// TwinCAT 3 PLC project LULSolarData
// ProgramVersion: 3.1.4020.10
// libraries:
//   Tc2_BA, * (Beckhoff Automation GmbH)
//   Tc2_EtherCAT, * (Beckhoff Automation GmbH)
//   Tc2_IoFunctions, * (Beckhoff Automation GmbH)
//   Tc2_ModbusRTU, * (Beckhoff Automation GmbH)
//   Tc2_ModbusSrv, * (Beckhoff Automation GmbH)
//   Tc2_SerialCom, * (Beckhoff Automation GmbH)
//   Tc2_Standard, * (Beckhoff Automation GmbH)
//   Tc2_SUPS, * (Beckhoff Automation GmbH)
//   Tc2_System, * (Beckhoff Automation GmbH)
//   Tc2_Utilities, * (Beckhoff Automation GmbH)
//   Tc3_IotBase, * (Beckhoff Automation GmbH)
//   Tc3_Module, * (Beckhoff Automation GmbH)
// project tree:
//   DUTs/Cluster Control/Huvudstrukt/ ST_ClusterCtrl.TcDUT
//   DUTs/Cluster Control/ ST_ActivePower.TcDUT, ST_ApparentPower.TcDUT, ST_DcCurrent.TcDUT, ST_LineCurrent.TcDUT, ST_LineVoltage.TcDUT, ST_PV_data.TcDUT, ST_ReactivePower.TcDUT, ST_Si420TC.TcDUT, ST_StatusCtrl.TcDUT, ST_Yield.TcDUT
//   DUTs/Hukseflux SR05/ ST_SR05_IrrMeter.TcDUT
//   DUTs/IoT/ U_Payload.TcDUT
//   DUTs/Schneider IEM/Huvudstrukt/ ST_IEM3255.TcDUT
//   DUTs/Schneider IEM/ ST_AlarmValue.TcDUT, ST_OverloadAL.TcDUT, ST_Current.TcDUT, ST_Frequency.TcDUT, ST_PartialEnergy.TcDUT, ST_PhaseEnergy.TcDUT, ST_Power.TcDUT, ST_Power2.TcDUT, ST_PowerFactor.TcDUT, ST_TotalEnergy.TcDUT, ST_Voltage.TcDUT, ST_Voltage2.TcDUT
//   DUTs/WXT530/Huvudstrukt/ ST_WXT530.TcDUT
//   DUTs/WXT530/ ST_WindData.TcDUT
//   GVLs/ GVL_ClusterCtrl.TcGVL, GVL_Fastighet.TcGVL, GVL_IO.TcGVL, GVL_IoT.TcGVL, GVL_Larm.TcGVL, GVL_MX41.TcGVL, GVL_SR05.TcGVL, GVL_WXT530.TcGVL
//   / Modbus.TcTTO, PlcTask.TcTTO
//   POUs/ClusterCtrl/ F15_ClusterCtrl.TcPOU, F15_ClusterCtrl_Larm.TcPOU
//   POUs/IO/ F15_AS3_AI.TcPOU
//   POUs/Loggning/ Cluster_Logg.TcPOU, Cluster_Logg_2.TcPOU, Cluster_Logg_3.TcPOU, Cluster_Sensor_Logg.TcPOU, FB_IoT_Publisher.TcPOU, iEM3255_Logg.TcPOU, MAIN_loggning.TcPOU, Temp_Logg.TcPOU, SR05_Logg.TcPOU, WXT530_Logg.TcPOU
//   POUs/ MAIN.TcPOU
//   POUs/MQ41/ F15_AS3_MQ41.TcPOU
//   POUs/Novram Hantering/ NovramHandling.TcPOU
//   POUs/Novram Hantering/ST_Novram/ ST_NovramData.TcDUT
//   POUs/Systemprogram/ PersistentData.TcPOU, PLC_Batteri_Larm.TcPOU, PLC_TID.TcPOU, WatchDog_PLC.TcPOU
//   POUs/WXT530/ F15_AS3_WXT530.TcPOU, RS485.TcPOU
//   POUs/_FBs/ AI_filter.TcPOU, ClusterControl_3Unit.TcPOU, FB_CountYears.TcPOU, FB_FL.TcPOU, FB_Pulsfilter.TcPOU, FB_SaveToCSV_ClusterCtrl.TcPOU, FB_SaveToCSV_SR05.TcPOU, FB_SaveToCSV_Schneider.TcPOU, FB_SaveToCSV_Cluster_Sensors.TcPOU, FB_SaveToCSV_Temp.TcPOU, FB_SaveToCSV_WXT530.TcPOU, FB_SCHNEIDER_iEM3150.TcPOU, FB_HUKSEFLUX_SR05.TcPOU, FB_WXT350.TcPOU, F_WordSwap.TcPOU
// real-time tasks:
//   TASK PlcTask: cycle T#5ms, priority 3, ADS port 350
//   TASK Modbus_seriell: cycle T#1ms, priority 1, ADS port 352
// I/O:
//   DEVICE Device 1 (EtherCAT), AmsNetId 172.17.204.1.2.1
//     Term 5 (EK1200) [EK1200-5000 EtherCAT Power supply (2A E-Bus)]
//       Term 6 (EL6021) [EL6021 Interface (RS422/485)]
//       Term 7 (EL6021) [EL6021 Interface (RS422/485)]
//       Box 8 (BK1250)
//   DEVICE Device 5 (USB) (disabled)
//   DEVICE Device 6 (NOV-DP-RAM)
// variable links:
//   LULSolarData/LULSolarData Instance <-> Device 1 (EtherCAT)/Term 5 (EK1200)/Box 8 (BK1250)
//     PlcTask Inputs/GVL_IO._AI1 <-> Term 2 (KL3208-0010-4)/Channel 1/Data In
//     PlcTask Inputs/GVL_IO._AI2 <-> Term 2 (KL3208-0010-4)/Channel 2/Data In
//     PlcTask Inputs/GVL_IO._AI3 <-> Term 2 (KL3208-0010-4)/Channel 3/Data In
//     PlcTask Inputs/GVL_IO._AI4 <-> Term 2 (KL3208-0010-4)/Channel 4/Data In
//     PlcTask Inputs/GVL_IO._AI5 <-> Term 3 (KL3208-0010-4)/Channel 1/Data In
//     PlcTask Inputs/GVL_IO._AI6 <-> Term 3 (KL3208-0010-4)/Channel 2/Data In
//     PlcTask Inputs/GVL_IO._AI7 <-> Term 3 (KL3208-0010-4)/Channel 3/Data In
//     PlcTask Inputs/GVL_IO._AI8 <-> Term 3 (KL3208-0010-4)/Channel 4/Data In
//   LULSolarData/LULSolarData Instance <-> Device 1 (EtherCAT)/Term 5 (EK1200)/Term 6 (EL6021)
//     Modbus Inputs/RS485.ComIn_Com1/D <-> COM TxPDO-Map Inputs/Data In 0
//     Modbus Inputs/RS485.ComIn_Com1/D @bit {8..168 step 8} <-> COM TxPDO-Map Inputs/Data In {1..21}  (21 links)
//     Modbus Inputs/RS485.ComIn_Com1/Status <-> COM TxPDO-Map Inputs/Status
//     Modbus Outputs/RS485.ComOut_Com1/Ctrl <-> COM RxPDO-Map Outputs/Ctrl
//     Modbus Outputs/RS485.ComOut_Com1/D <-> COM RxPDO-Map Outputs/Data Out 0
//     Modbus Outputs/RS485.ComOut_Com1/D @bit {8..168 step 8} <-> COM RxPDO-Map Outputs/Data Out {1..21}  (21 links)
//   LULSolarData/LULSolarData Instance <-> Device 1 (EtherCAT)/Term 5 (EK1200)/Term 7 (EL6021)
//     Modbus Inputs/F15_AS3_MQ41.Energimatare.fbRtuMaster.InData/D <-> COM TxPDO-Map Inputs/Data In 0
//     Modbus Inputs/F15_AS3_MQ41.Energimatare.fbRtuMaster.InData/D @bit {8..168 step 8} <-> COM TxPDO-Map Inputs/Data In {1..21}  (21 links)
//     Modbus Inputs/F15_AS3_MQ41.Energimatare.fbRtuMaster.InData/Status <-> COM TxPDO-Map Inputs/Status
//     Modbus Outputs/F15_AS3_MQ41.Energimatare.fbRtuMaster.OutData/Ctrl <-> COM RxPDO-Map Outputs/Ctrl
//     Modbus Outputs/F15_AS3_MQ41.Energimatare.fbRtuMaster.OutData/D <-> COM RxPDO-Map Outputs/Data Out 0
//     Modbus Outputs/F15_AS3_MQ41.Energimatare.fbRtuMaster.OutData/D @bit {8..168 step 8} <-> COM RxPDO-Map Outputs/Data Out {1..21}  (21 links)

CONFIGURATION LULSolarData
    RESOURCE PLC ON TwinCAT3
        TASK Modbus(INTERVAL := T#1ms, PRIORITY := 1);
        TASK PlcTask(INTERVAL := T#5ms, PRIORITY := 3);
        PROGRAM F15_AS3_MQ41 WITH Modbus : F15_AS3_MQ41;
        PROGRAM F15_AS3_WXT530 WITH Modbus : F15_AS3_WXT530;
        PROGRAM RS485 WITH Modbus : RS485;
        PROGRAM MAIN WITH PlcTask : MAIN;
    END_RESOURCE
END_CONFIGURATION

// ---- DUTs/Cluster Control/Huvudstrukt/ST_ClusterCtrl.TcDUT
TYPE ST_ClusterCtrl :
STRUCT
	stActivePower			:ST_ActivePower;
	stLineVoltage			:ST_LineVoltage;
	stLineCurrent			:ST_LineCurrent;
	stYield					:ST_Yield;
	stPVDATA				:ST_PV_data;
	stStatus				:ST_StatusCtrl;
	stReactivePower			:ST_ReactivePower;
	stApparentPower			:ST_ApparentPower;
	stSi420					:ST_Si420TC;
	nTotEnergyConsInternally:DWORD;
	nInverterInteriorTemp 	:DWORD;
	nEnergySavingMode		:DWORD;
END_STRUCT
END_TYPE

// ---- DUTs/Cluster Control/ST_ActivePower.TcDUT
TYPE ST_ActivePower :
STRUCT
	
	ActivePower_Total		:DINT;
	ActivePower_L1			:DINT;
	ActivePower_L2			:DINT;
	ActivePower_L3			:DINT;
	
END_STRUCT
END_TYPE

// ---- DUTs/Cluster Control/ST_ApparentPower.TcDUT
TYPE ST_ApparentPower :
STRUCT
	ApparentPower_Total			:DINT;
	ApparentPower_L1			:DINT;
	ApparentPower_L2			:DINT;
	ApparentPower_L3			:DINT;
END_STRUCT
END_TYPE

// ---- DUTs/Cluster Control/ST_DcCurrent.TcDUT
TYPE ST_DcCurrent :
STRUCT
	
END_STRUCT
END_TYPE

// ---- DUTs/Cluster Control/ST_LineCurrent.TcDUT
TYPE ST_LineCurrent :
STRUCT
	
	LineCurrent_Total		:DWORD;
	LineCurrent_L1			:DWORD;
	LineCurrent_L2			:DWORD;
	LineCurrent_L3			:DWORD;
	PowerFrequency			:DWORD;
	
END_STRUCT
END_TYPE

// ---- DUTs/Cluster Control/ST_LineVoltage.TcDUT
TYPE ST_LineVoltage :
STRUCT
	
	LineVoltage_L1_N 	:DWORD;
	LineVoltage_L2_N 	:DWORD;
	LineVoltage_L3_N 	:DWORD;
	LineVoltage_L1_L2 	:DWORD;
	LineVoltage_L2_L3 	:DWORD;
	LineVoltage_L3_L1 	:DWORD;
	
END_STRUCT
END_TYPE

// ---- DUTs/Cluster Control/ST_PV_data.TcDUT
TYPE ST_PV_data :
STRUCT
	Line_current_L1		:DINT;
	Line_current_L2		:DINT;
	Line_current_L3		:DINT;
	PV_Power			:DWORD;
END_STRUCT
END_TYPE

// ---- DUTs/Cluster Control/ST_ReactivePower.TcDUT
TYPE ST_ReactivePower :
STRUCT
	ReactivePower_Total		:DINT;
	ReactivePower_L1		:DINT;
	ReactivePower_L2		:DINT;
	ReactivePower_L3		:DINT;
END_STRUCT
END_TYPE

// ---- DUTs/Cluster Control/ST_Si420TC.TcDUT
TYPE ST_Si420TC :
STRUCT
	Irradiation	:DINT;
END_STRUCT
END_TYPE

// ---- DUTs/Cluster Control/ST_StatusCtrl.TcDUT
TYPE ST_StatusCtrl :
STRUCT
	Device_Status		:DWORD;
END_STRUCT
END_TYPE

// ---- DUTs/Cluster Control/ST_Yield.TcDUT
TYPE ST_Yield :
STRUCT
	Total_AC_energy_all_conductors_Wh		:DWORD;
	Total_AC_energy_all_conductors_kWh		:DWORD;
	Total_AC_energy_all_conductors_MWh		:DWORD;
	Energy_current_day_all_conductors_Wh	:DWORD;
	Energy_current_day_all_conductors_kWh	:DWORD;
	Energy_current_day_all_conductors_MWh	:DWORD;
	Operating_time							:DWORD;
	Feed_in_time							:DWORD;	
END_STRUCT
END_TYPE

// ---- DUTs/Hukseflux SR05/ST_SR05_IrrMeter.TcDUT
TYPE ST_SR05_IrrMeter :
STRUCT
	Solar_Irradiance_raw:  		REAL;
	Solar_Irradiance:   		REAL;
	Sensor_Body_Temp:			REAL;
	Sensor_Elec_Resistance:		REAL;
	Sensor_voltage_output:		REAL;
	
END_STRUCT
END_TYPE

// ---- DUTs/IoT/U_Payload.TcDUT
TYPE U_Payload :
UNION
	sPayload : STRING(3999);
	aPayload : ARRAY[0..3999] OF BYTE;
END_UNION
END_TYPE

// ---- DUTs/Schneider IEM/Huvudstrukt/ST_IEM3255.TcDUT
TYPE ST_IEM3255 :
STRUCT
	stCurrent:			ST_Current;
	stVolt:				ST_Voltage;
	stVolt2:			ST_Voltage2;
	stPower:			ST_Power;
	stPower2:			ST_Power2;
	stPowerFactor:		ST_PowerFactor;
	stFrequency:		ST_Frequency;
	stTotalEnergy:		ST_TotalEnergy;
	stPartialEnergy:	ST_PartialEnergy;
	stPhaseEnergy:		ST_PhaseEnergy;
	stOverloadAL:		ST_OverloadAL;
	stAlarmValue:		ST_AlarmValue;
END_STRUCT
END_TYPE

// ---- DUTs/Schneider IEM/ST_AlarmValue.TcDUT
TYPE ST_AlarmValue :
STRUCT
	Last_Alarm_Value:	REAL;
END_STRUCT
END_TYPE

// ---- DUTs/Schneider IEM/ST_OverloadAL.TcDUT
TYPE ST_OverloadAL :
STRUCT
	Status:	BIT;
END_STRUCT
END_TYPE

// ---- DUTs/Schneider IEM/ST_Current.TcDUT
TYPE ST_Current :
STRUCT
	Phase_1_current:	REAL;
	Phase_2_current:	REAL;
	Phase_3_current:	REAL;
END_STRUCT
END_TYPE

// ---- DUTs/Schneider IEM/ST_Frequency.TcDUT
TYPE ST_Frequency :
STRUCT
	Frequency:	REAL;
END_STRUCT
END_TYPE

// ---- DUTs/Schneider IEM/ST_PartialEnergy.TcDUT
TYPE ST_PartialEnergy :
STRUCT
	Partial_Active_Energy_Import:	REAL;
	Partial_Reactive_Energy_Import:	REAL;
END_STRUCT
END_TYPE

// ---- DUTs/Schneider IEM/ST_PhaseEnergy.TcDUT
TYPE ST_PhaseEnergy :
STRUCT
	Active_Energy_Import_Phase_1:	REAL;
	Active_Energy_Import_Phase_2:	REAL;
	Active_Energy_Import_Phase_3:	REAL;
END_STRUCT
END_TYPE

// ---- DUTs/Schneider IEM/ST_Power.TcDUT
TYPE ST_Power :
STRUCT
	Active_Power_Phase_1:	REAL;
	Active_Power_Phase_2:	REAL;
	Active_Power_Phase_3:	REAL;
	Total_Active_Power:		REAL;
END_STRUCT
END_TYPE

// ---- DUTs/Schneider IEM/ST_Power2.TcDUT
TYPE ST_Power2 :
STRUCT
	Total_Reactive_Power:	REAL;
	Reserved2:				REAL;
	Reserved3:				REAL;
	Reserved4:				REAL;
	Total_Apparent_Power:	REAL;

END_STRUCT
END_TYPE

// ---- DUTs/Schneider IEM/ST_PowerFactor.TcDUT
TYPE ST_PowerFactor :
STRUCT
	Total_Power_Factor:	REAL;
END_STRUCT
END_TYPE

// ---- DUTs/Schneider IEM/ST_TotalEnergy.TcDUT
TYPE ST_TotalEnergy :
STRUCT
	Total_Active_Energy_Import:		REAL;
	Total_Active_Energy_Export:		REAL;
	Total_Reactive_Energy_Import:	REAL;
	Total_Reactive_Energy_Export:	REAL;
END_STRUCT
END_TYPE

// ---- DUTs/Schneider IEM/ST_Voltage.TcDUT
TYPE ST_Voltage :
STRUCT
	Voltage_L1_L2:	REAL;
	Voltage_L2_L3:	REAL;
	Voltage_L3_L1:	REAL;	
END_STRUCT
END_TYPE

// ---- DUTs/Schneider IEM/ST_Voltage2.TcDUT
TYPE ST_Voltage2 :
STRUCT
	Voltage_L1_N:	REAL;
	Voltage_L2_N:	REAL;
	Voltage_L3_N:	REAL;
END_STRUCT
END_TYPE

// ---- DUTs/WXT530/Huvudstrukt/ST_WXT530.TcDUT
TYPE ST_WXT530 :
STRUCT
	stWindData			:ST_WindData;
END_STRUCT
END_TYPE

// ---- DUTs/WXT530/ST_WindData.TcDUT
TYPE ST_WindData :
STRUCT

Dn	:REAL;  (*Wind direction minimum (D = degrees)*)
Dm	:REAL;  (*Wind direction average (D = degrees)*)
Dx	:REAL;  (*Wind direction maximum (D = degrees*)
Sn	:REAL;  (*Wind speed minimum (M = m/S)*)
Sm	:REAL;  (*Wind speed average (M = m/S)*)
Sx	:REAL;  (*Wind speed maximum (M = m/S)*)	

END_STRUCT
END_TYPE

// ---- POUs/Novram Hantering/ST_Novram/ST_NovramData.TcDUT
TYPE ST_NovramData :
STRUCT
END_STRUCT
END_TYPE

// ---- GVLs/GVL_ClusterCtrl.TcGVL
{attribute 'qualified_only'}
VAR_GLOBAL	
		
_CCtrl_V1_IT				AT%MX2000.0			:BOOL;  	(* Driftindikering *)
_CCtrl_V1_P					AT%MB2004			:REAL;  	(* Total momentan effekt *)
_CCtrl_V1_P1				AT%MB2008			:REAL;  	(* Effekt L1 *)
_CCtrl_V1_P2				AT%MB2012			:REAL;  	(* Effekt L2 *)
_CCtrl_V1_P3				AT%MB2016			:REAL;  	(* Effekt L3 *)
_CCtrl_V1_U1_L1_N			AT%MB2020			:REAL;  	(* Spänning L1-N *)
_CCtrl_V1_U2_L2_N			AT%MB2024			:REAL;  	(* Spänning L2-N *)
_CCtrl_V1_U3_L3_N			AT%MB2028			:REAL;  	(* Spänning L3-N *)
_CCtrl_V1_U1_L1_L2			AT%MB2032			:REAL;  	(* Spänning L1-L2*)
_CCtrl_V1_U2_L2_L3			AT%MB2036			:REAL;  	(* Spänning L2-L3 *)
_CCtrl_V1_U3_L3_L1			AT%MB2040			:REAL;  	(* Spänning L3-L1 *)
_CCtrl_V1_Itot									:REAL; 		(* Total Ström L1,L2,L3*)
_CCtrl_V1_I1				AT%MB2044			:REAL;  	(* Ström L1 *)
_CCtrl_V1_I2				AT%MB2048			:REAL;  	(* Ström L2 *)
_CCtrl_V1_I3				AT%MB2052			:REAL;  	(* Ström L3 *)
_CCtrl_V1_Yield_Wh			AT%MB2056			:REAL;  	(* Total avkastning Wh *)
_CCtrl_V1_Yield_kWh			AT%MB2060			:REAL;  	(* Total avkastning kWh *)
_CCtrl_V1_Yield_MWh			AT%MB2064			:REAL;  	(* Total avkastning MWh *)
_CCtrl_V1_YieldDay_Wh		AT%MB2068			:REAL;  	(* Total avkastning aktuell dag Wh *)
_CCtrl_V1_YieldDay_kWh		AT%MB2072			:REAL;  	(* Total avkastning aktuell dag kWh *)
_CCtrl_V1_PV				AT%MB2076			:REAL;  	(* PV effekt*)
_CCtrl_V1_HZ				AT%MB2080			:REAL;  	(* Frekvens *)	
_CCtrl_V1_TECInt								:REAL;		(* Total Energy Consumed Internally i växelriktaren *)	
_CCtrl_V1_APtot									:REAL;		(* Total Apparent Power L1,L2,L3*)
_CCtrl_V1_AP1									:REAL;  	(* Apparent Power L1 *)
_CCtrl_V1_AP2									:REAL;  	(* Apparent Power L2 *)
_CCtrl_V1_AP3									:REAL;  	(* Apparent Power L3 *)
_CCtrl_V1_RPtot									:REAL;		(* Total Reactive Power L1,L2,L3*)
_CCtrl_V1_RP1									:REAL;  	(* Reactive Power L1 *)
_CCtrl_V1_RP2									:REAL;  	(* Reactive Power L2 *)
_CCtrl_V1_RP3									:REAL;  	(* Reactive Power L3 *)
_CCtrl_V1_EnSaveMode							:REAL;		(* Energy Saving Mode Switched On (1129=Yes, 1130=No) *)

							
_CCtrl_V2_IT				AT%MX2400.0			:BOOL;  	(* Driftindikering *)
_CCtrl_V2_P					AT%MB2404			:REAL;  	(* Total momentan effekt *)
_CCtrl_V2_P1				AT%MB2408			:REAL;  	(* Effekt L1 *)
_CCtrl_V2_P2				AT%MB2412			:REAL;  	(* Effekt L2 *)
_CCtrl_V2_P3				AT%MB2416			:REAL;  	(* Effekt L3 *)
_CCtrl_V2_U1_L1_N			AT%MB2420			:REAL;  	(* Spänning L1-N *)
_CCtrl_V2_U2_L2_N			AT%MB2424			:REAL;  	(* Spänning L2-N *)
_CCtrl_V2_U3_L3_N			AT%MB2428			:REAL;  	(* Spänning L3-N *)
_CCtrl_V2_U1_L1_L2			AT%MB2432			:REAL;  	(* Spänning L1-L2*)
_CCtrl_V2_U2_L2_L3			AT%MB2436			:REAL;  	(* Spänning L2-L3 *)
_CCtrl_V2_U3_L3_L1			AT%MB2440			:REAL;  	(* Spänning L3-L1 *)
_CCtrl_V2_Itot									:REAL; 		(* Total Ström L1,L2,L3*)
_CCtrl_V2_I1				AT%MB2444			:REAL;  	(* Ström L1 *)
_CCtrl_V2_I2				AT%MB2448			:REAL;  	(* Ström L2 *)
_CCtrl_V2_I3				AT%MB2452			:REAL;  	(* Ström L3 *)
_CCtrl_V2_Yield_Wh			AT%MB2456			:REAL;  	(* Total avkastning Wh *)
_CCtrl_V2_Yield_kWh			AT%MB2460			:REAL;  	(* Total avkastning kWh *)
_CCtrl_V2_Yield_MWh			AT%MB2464			:REAL;  	(* Total avkastning MWh *)
_CCtrl_V2_YieldDay_Wh		AT%MB2468			:REAL;  	(* Total avkastning aktuell dag Wh *)
_CCtrl_V2_YieldDay_kWh		AT%MB2472			:REAL;  	(* Total avkastning aktuell dag kWh *)
_CCtrl_V2_PV				AT%MB2476			:REAL;  	(* PV effekt*)
_CCtrl_V2_HZ				AT%MB2480			:REAL;  	(* Frekvens *)		
_CCtrl_V2_TECInt								:REAL;		(* Total Energy Consumed Internally i växelriktaren *)					
_CCtrl_V2_APtot									:REAL;		(* Total Apparent Power L1,L2,L3*)
_CCtrl_V2_AP1									:REAL;  	(* Apparent Power L1 *)
_CCtrl_V2_AP2									:REAL;  	(* Apparent Power L2 *)
_CCtrl_V2_AP3									:REAL;  	(* Apparent Power L3 *)
_CCtrl_V2_RPtot									:REAL;		(* Total Reactive Power L1,L2,L3*)
_CCtrl_V2_RP1									:REAL;  	(* Reactive Power L1 *)
_CCtrl_V2_RP2									:REAL;  	(* Reactive Power L2 *)
_CCtrl_V2_RP3									:REAL;  	(* Reactive Power L3 *)
_CCtrl_V2_EnSaveMode							:REAL;		(* Energy Saving Mode Switched On (1129=Yes, 1130=No) *)
							
_CCtrl_V3_IT				AT%MX2800.0			:BOOL;  	(* Driftindikering *)
_CCtrl_V3_P					AT%MB2804			:REAL;  	(* Total momentan effekt *)
_CCtrl_V3_P1				AT%MB2808			:REAL;  	(* Effekt L1 *)
_CCtrl_V3_P2				AT%MB2812			:REAL;  	(* Effekt L2 *)
_CCtrl_V3_P3				AT%MB2816			:REAL;  	(* Effekt L3 *)
_CCtrl_V3_U1_L1_N			AT%MB2820			:REAL;  	(* Spänning L1-N *)
_CCtrl_V3_U2_L2_N			AT%MB2824			:REAL;  	(* Spänning L2-N *)
_CCtrl_V3_U3_L3_N			AT%MB2828			:REAL;  	(* Spänning L3-N *)
_CCtrl_V3_U1_L1_L2			AT%MB2832			:REAL;  	(* Spänning L1-L2*)
_CCtrl_V3_U2_L2_L3			AT%MB2836			:REAL;  	(* Spänning L2-L3 *)
_CCtrl_V3_U3_L3_L1			AT%MB2840			:REAL;  	(* Spänning L3-L1 *)
_CCtrl_V3_Itot									:REAL; 		(* Total Ström L1,L2,L3*)
_CCtrl_V3_I1				AT%MB2844			:REAL;  	(* Ström L1 *)
_CCtrl_V3_I2				AT%MB2848			:REAL;  	(* Ström L2 *)
_CCtrl_V3_I3				AT%MB2852			:REAL;  	(* Ström L3 *)
_CCtrl_V3_Yield_Wh			AT%MB2856			:REAL;  	(* Total avkastning Wh *)
_CCtrl_V3_Yield_kWh			AT%MB2860			:REAL;  	(* Total avkastning kWh *)
_CCtrl_V3_Yield_MWh			AT%MB2864			:REAL;  	(* Total avkastning MWh *)
_CCtrl_V3_YieldDay_Wh		AT%MB2868			:REAL;  	(* Total avkastning aktuell dag Wh *)
_CCtrl_V3_YieldDay_kWh		AT%MB2872			:REAL;  	(* Total avkastning aktuell dag kWh *)
_CCtrl_V3_PV				AT%MB2876			:REAL;  	(* PV effekt*)
_CCtrl_V3_HZ				AT%MB2880			:REAL;  	(* Frekvens *)
_CCtrl_V3_TECInt								:REAL;		(* Total Energy Consumed Internally i växelriktaren *)
_CCtrl_V3_APtot									:REAL;		(* Total Apparent Power L1,L2,L3*)
_CCtrl_V3_AP1									:REAL;  	(* Apparent Power L1 *)
_CCtrl_V3_AP2									:REAL;  	(* Apparent Power L2 *)
_CCtrl_V3_AP3									:REAL;  	(* Apparent Power L3 *)
_CCtrl_V3_RPtot									:REAL;		(* Total Reactive Power L1,L2,L3*)
_CCtrl_V3_RP1									:REAL;  	(* Reactive Power L1 *)
_CCtrl_V3_RP2									:REAL;  	(* Reactive Power L2 *)
_CCtrl_V3_RP3									:REAL;  	(* Reactive Power L3 *)
_CCtrl_V3_EnSaveMode							:REAL;		(* Energy Saving Mode Switched On (1129=Yes, 1130=No) *)

_CCtrl_ST_Si420TC								:REAL:		(*IMT irr meter behövs fler*)	
END_VAR

// ---- GVLs/GVL_Fastighet.TcGVL
{attribute 'qualified_only'}
VAR_GLOBAL PERSISTENT
	FastighetsBeteckning : STRING := 'A1157_AS3';
	
	(* Microsoft Azure IoT Hub Settings *)
	//IoTHostName			 : STRING := 'sole-ap-01.lul-net.ad.lul.se';
	IoTHostName			 : STRING := '172.23.10.77'; (* <- Will not be used in vaksala*)
	IoTHostPort 		 : UINT	:= 1883;	(* <- Will not be used in vaksala*)
	IoTTopicPub 		 : STRING := 'devices/TestPlc/messages/events/readpipe/';
	PublishTime 		 : TIME := T#15S; //OBS!! Väderstationens värden samt analoga givare rapporteras till IoT var 4e ggn - se FB_IoT_Publisher och case 10
	
	(* Aktivering/deaktivering av enheter *)
	EnergyMeter			: BOOL := TRUE; //Schneider iEM3255 Energimätare
	IO 					: BOOL := TRUE; //Analoga mätvärden
	WXT530				: BOOL := TRUE; //Väderstation Vaisala modell WXT530 
	SMAClusterCntrl		: BOOL := TRUE; //SMA CLusterControler, använd för att samla ihop fler Växelriktare i en kommunikationspunkt
	
	//Si420TC				: BOOL := TRUE; //Den andra solinstrålningsmätaren
	SR05				: BOOL := TRUE; //Solinstrålningsgivare Hukseflux SR05
		
END_VAR
VAR_GLOBAL
	(* Loggning - csv fil sparas lokalt på datorn*)
	CSVClusterCtrl		: BOOL := TRUE; //Växelriktare sammankopplade med en SMA Cluster Controler
	CSVEnergyMeter		: BOOL := TRUE; //Energimätare Schneider iEM3255
	CSVTempProbes		: BOOL := TRUE; //Tempgivare solpaneler, analog input
	CSVWXT530			: BOOL := TRUE; //Väderstation Vaisala modell WXT530
	CSVSR05				: BOOL := TRUE; //SOLINSTRÅLINGS MÄTARE
	//CSVSi420TC			: BOOL:=TRUE // Andra solisntrålningsmätaren kisel
END_VAR

// ---- GVLs/GVL_IO.TcGVL
{attribute 'qualified_only'}
VAR_GLOBAL
(* PLC Year/Month/Day/Time *)									
	_PLC_YY			AT%MB50				:WORD;			(* Aktuellt år i PLC *)	
	_PLC_MM			AT%MB52				:WORD;			(* Aktuell månad i PLC *)		
	_PLC_DD			AT%MB54				:WORD;			(* Aktuell dag i PLC *)	
	_PLC_HHMM		AT%MB56				:WORD;			(* Aktuell tid i PLC *)		
											
(*Analoga in, hårdvara*)									
	_AI1			AT%IB100			 :INT;			(*Kalibrerat mätvärde*)
	_AI2			AT%IB102			 :INT;			(*Kalibrerat mätvärde*)
	_AI3			AT%IB104			 :INT;			(*Kalibrerat mätvärde*)
	_AI4			AT%IB106			 :INT;			(*Kalibrerat mätvärde*)
	_AI5			AT%IB108			 :INT;			(*Kalibrerat mätvärde*)
	_AI6			AT%IB110			 :INT;			(*Kalibrerat mätvärde*)
	_AI7			AT%IB112			 :INT;			(*Kalibrerat mätvärde*)
	_AI8			AT%IB114			 :INT;			(*Kalibrerat mätvärde*)
																																																																																								
(*Analoga in*)										
	_GT41_MV 		AT%MB100			 :INT;			(*Kalibrerat mätvärde*)
	_GT42_MV 		AT%MB102			 :INT;			(*Kalibrerat mätvärde*)
	_GT43_MV 		AT%MB104			 :INT;			(*Kalibrerat mätvärde*)
	_GT44_MV 		AT%MB106			 :INT;			(*Kalibrerat mätvärde*)
	_GT45_MV 		AT%MB108			 :INT;			(*Kalibrerat mätvärde*)
	_GT46_MV 		AT%MB110			 :INT;			(*Kalibrerat mätvärde*)
	_GT47_MV 		AT%MB112			 :INT;			(*Kalibrerat mätvärde*)
	_GT48_MV 		AT%MB114			 :INT;			(*Kalibrerat mätvärde*)

END_VAR

// ---- GVLs/GVL_IoT.TcGVL
{attribute 'qualified_only'}
VAR_GLOBAL PERSISTENT
	uPayloadQueue : ARRAY[0..nMaxPayloadBuffer] OF U_Payload;
	nLastPos : INT;
	bBufferFull : BOOL;
	bBufferEmpty : BOOL;
	nTotalMessagePublished : ULINT;
END_VAR
VAR_GLOBAL CONSTANT
	nMaxPayloadBuffer : INT := 100;
END_VAR
VAR_GLOBAL
	uPayloadEmpty : U_Payload;
END_VAR

// ---- GVLs/GVL_Larm.TcGVL
{attribute 'qualified_only'}
VAR_GLOBAL

	(* Larmtaggar *)								
	_BATT_L			AT%MX5000.0			:BOOL;  		(* Låg batterispänning *)
	_PLC_WD			AT%MX5000.1			:BOOL;  		(* Watchdog *)
	_MX41_LC			AT%MX5000.2			:BOOL;  		(* Kommunikationsfel*)
	_GW3U_LC			AT%MX5000.3			:BOOL;  		(* Kommunikationsfel*)
	_CCtrl_LC			AT%MX5000.4			:BOOL;  		(* Kommunikationsfel*)
	_CCtrl_V1_L		AT%MX5000.5			:BOOL;  		(* Summalarm *)
	_CCtrl_V1_LM		AT%MX5000.6			:BOOL;  		(* Omriktare frånslagen *)
	_CCtrl_V2_L		AT%MX5000.7			:BOOL;  		(* Summalarm *)
	_CCtrl_V2_LM		AT%MX5001.0			:BOOL;  		(* Omriktare frånslagen *)
	_CCtrl_V3_L		AT%MX5001.1			:BOOL;  		(* Summalarm *)
	_CCtrl_V3_LM		AT%MX5001.2			:BOOL;  		(* Omriktare frånslagen *)
	
	
	
	_BATT_L_ACK		AT%MX5030.0			:BOOL;  		(* Ack batterilarm *)

							
								
END_VAR					
								
VAR_GLOBAL PERSISTENT								
								
								
(* Larminställningar *)								
	_MX41_LC_FL		AT%MB5104			:INT;  			(* Larmfördröjning *)
	_GW3U_LC_FL		AT%MB5106			:INT;  			(* Larmfördröjning *)
	_CCtrl_LC_FL		AT%MB5108			:INT;  			(* Larmfördröjning *)
	_CCtrl_V1_L_FL		AT%MB5110			:INT;  			(* Larmfördröjning *)
	_CCtrl_V2_L_FL		AT%MB5114			:INT;  			(* Larmfördröjning *)
	_CCtrl_V3_L_FL		AT%MB5118			:INT;  			(* Larmfördröjning *)
	

END_VAR

// ---- GVLs/GVL_MX41.TcGVL
{attribute 'qualified_only'}
VAR_GLOBAL	
																					
(*Mätvärden*)											
_I1 				AT%MB300			:REAL;			(*Ström i Ampere fas 1, adr 3000*)
_I2					AT%MB304			:REAL;			(*Ström i Ampere fas 2, adr 3002*)
_I3					AT%MB308			:REAL;			(*Ström i Ampere fas 3, adr 3004*)
					
_U1_U2				AT%MB312			:REAL;			(*Spänning L1-L2 i Volt, adr 3020*)
_U2_U3				AT%MB316			:REAL;			(*Spänning L2-L3 i Volt, adr 3022*)
_U3_U1				AT%MB320			:REAL;			(*Spänning L3-L1  i Volt, adr 3024*)
					
_U1_N				AT%MB324			:REAL;			(*Spänning L1-N i Volt, adr 3020*)
_U2_N				AT%MB328			:REAL;			(*Spänning L3-N i Volt, adr 3022*)
_U3_N				AT%MB332			:REAL;			(*Spänning L2-N i Volt, adr 3024*)
					
_P1					AT%MB336			:REAL;			(*Effekt fas 1 i kW, adr 3054*)
_P2					AT%MB340			:REAL;			(*Effekt fas 2 i kW, adr 3056*)
_P3					AT%MB344			:REAL;			(*Effekt fas 3 i kW, adr 3058*)
					
_P					AT%MB348			:REAL;			(*Total aktiv effekt i kW, adr 3060*)
_PVAR				AT%MB352			:REAL;			(*Total reaktiv effekt i kVAR, adr 3068*)
_PVA				AT%MB356			:REAL;			(*Total apparent effekt i kVA, adr 3076*)
					
_Pfa				AT%MB360			:REAL;			(*Effektfaktor , adr 3084*)
					
_HZ					AT%MB364			:REAL;			(*Effektfaktor , adr 3110*)
					
_WHAI				AT%MB368			:REAL;			(*Total aktiv energi import i Wh, adr 3204*)
_WHAE				AT%MB372			:REAL;			(*Total aktiv energi export i Wh, adr 3208*)
_VARHI				AT%MB376			:REAL;			(*Total reaktiv energi import i VARh, adr 3220*)
_VARHE				AT%MB380			:REAL;			(*Total reaktiv energi export i VARh, adr 3224*)
					
_WHPAI				AT%MB384			:REAL;			(*Partial aktiv energi import i Wh, adr 3256*)
_WHPAE				AT%MB388			:REAL;			(*Partial reaktiv energi import i Wh, adr 3272*)
					
_WHAEI1				AT%MB392			:REAL;			(*Aktiv energi import i Wh fas 1, adr 3518*)
_WHAEI2				AT%MB396			:REAL;			(*Aktiv energi import i Wh fas 2, adr 3522*)
_WHAEI3				AT%MB400			:REAL;			(*Aktiv energi import i Wh fas 3, adr 3526*)
					

END_VAR

// ---- GVLs/GVL_SR05.TcGVL
{attribute 'qualified_only'}
VAR_GLOBAL	
																					
(*Mätvärden*)											
_SolarIrr				:REAL;			(*Solar Irradiance, signal in x 0.01 W/m², adr 2+3*)
_BodyTemp				:REAL;			(*Sensor body temperature in x 0.01 °C, adr 6*)
_ElecResistance			:REAL;			(*Sensor electrical resistance in x 0.1 Ω, adr 7*)	
_VoltageOutput			:REAL;			(*Solar Irradiance, signal in x 0.01 W/m², adr 2+3*)


END_VAR

// ---- GVLs/GVL_WXT530.TcGVL
{attribute 'qualified_only'}
VAR_GLOBAL
	TxBuffer_Com1: ComBuffer;
	RxBuffer_Com1: ComBuffer;
										
(*Vind (aR1)*)								
	_GW3U_DN		AT%MB1000			:REAL;  		(*Vindriktning MIN, grader*)
	_GW3U_DM		AT%MB1004			:REAL;  		(*Vindriktning medel, grader*)
	_GW3U_DX		AT%MB1008			:REAL;  		(*Vindriktning MAX, grader*)
	_GW3U_SN		AT%MB1012			:REAL;  		(*Vindhastighet MIN, m/s*)
	_GW3U_SM		AT%MB1016			:REAL;  		(*Vindhastighet medel, m/s*)
	_GW3U_SX		AT%MB1020			:REAL;  		(*Vindhastighet MAX, m/s*)
											
(*Tryck, temperatur and fuktighet (aR2)*)								
	_GW3U_GT3U		AT%MB1024			:REAL;  		(*Utetemperatur,°C*)
	_GW3U_GT41 		AT%MB1028			:REAL;  		(*Intern temperatur °C*)
	_GW3U_GM41		AT%MB1032			:REAL;  		(*Relativ fuktighet, % RH*)
	_GW3U_GP41		AT%MB1036			:REAL;  		(*Lufttryck, hPa*)
																	
(*Nederbörd (aR3)*)								
	_GW3U_RC		AT%MB1040			:REAL;  		(*Regn ackumulerat, mm*)
	_GW3U_RD		AT%MB1044			:REAL;  		(*Regn varaktighet,  S*)
	_GW3U_RI		AT%MB1048			:REAL;  		(*Regn intensitet, mm/h*)
	_GW3U_HC		AT%MB1052			:REAL;  		(*Hagel accumulation, nedslag/cm2*)
	_GW3U_HD		AT%MB1056			:REAL;  		(*Hagel varkatighet, S*)
	_GW3U_HI 		AT%MB1060			:REAL;  		(*Hagel intensitet, nedslag/cm2h*)
	_GW3U_RP		AT%MB1064			:REAL;  		(*Regn peak intensitet, mm/h*)
	_GW3U_HP		AT%MB1068			:REAL;  		(*Hagelpeak intensitet, nedslag/cm2h*)
	
END_VAR

// ---- POUs/MQ41/F15_AS3_MQ41.TcPOU
PROGRAM F15_AS3_MQ41
VAR
	Energimatare: FB_SCHNEIDER_iEM3150;
	tof_0: TOF;

	FB_FL0: FB_FL;
END_VAR


// PAGE
GVL_Larm._MX41_LC := FB_FL0.Larm_ut;
tof_0(IN := Energimatare.bMbCommErr, PT := T#10s); // TOF
GVL_MX41._I2 := Energimatare._rI2;
GVL_MX41._I3 := Energimatare._rI3;
GVL_MX41._U1_U2 := Energimatare._rU_L1_L2;
GVL_MX41._U2_U3 := Energimatare._rU_L2_L3;
GVL_MX41._U3_U1 := Energimatare._rU_L3_L1;
GVL_MX41._U1_N := Energimatare._rU_L1_N;
GVL_MX41._U2_N := Energimatare._rU_L2_N;
GVL_MX41._U3_N := Energimatare._rU_L3_N;
GVL_MX41._P2 := Energimatare._rP2;
GVL_MX41._P3 := Energimatare._rP3;
GVL_MX41._P1 := Energimatare._rP1;
GVL_MX41._P := Energimatare._rPtot;
GVL_MX41._PVAR := Energimatare._rPVAR;
GVL_MX41._I1 := Energimatare._rI1;
Energimatare(bEnable := GVL_Fastighet.EnergyMeter, bySlaveAdr := 1); // FB_SCHNEIDER_iEM3150
GVL_MX41._PVA := Energimatare._rPVA;
GVL_MX41._Pfa := Energimatare._rPfa;
GVL_MX41._HZ := Energimatare._rHZ;
GVL_MX41._WHAI := Energimatare._rWHAI;
GVL_MX41._WHAE := Energimatare._rWHAE;
GVL_MX41._VARHI := Energimatare._rVARHI;
GVL_MX41._VARHE := Energimatare._rVARHE;
GVL_MX41._WHPAI := Energimatare._rWHPAI;
GVL_MX41._WHPAE := Energimatare._rWHPAE;
GVL_MX41._WHAEI1 := Energimatare._rWHAEI1;
GVL_MX41._WHAEI2 := Energimatare._rWHAEI2;
GVL_MX41._WHAEI3 := Energimatare._rWHAEI3;
FB_FL0(Larm_in := tof_0.Q, TID_in := GVL_Larm._MX41_LC_FL); // FB_FL

END_PROGRAM

// ---- POUs/_FBs/FB_SCHNEIDER_iEM3150.TcPOU

FUNCTION_BLOCK FB_SCHNEIDER_iEM3150
VAR_INPUT
	bEnable:			BOOL;		(*Enable*)
	bySlaveAdr:			BYTE;		(*Slav Id*)
END_VAR
VAR_OUTPUT
	bBusy:					BOOL;		(*Upptagen med arbete*)
	bMbCommErr:				BOOL;		(*Modbus Komm. fel*)
	
	_rI1 				:REAL;			(*Ström i Ampere fas 1, adr 3000*)
	_rI2				:REAL;			(*Ström i Ampere fas 2, adr 3002*)
	_rI3				:REAL;			(*Ström i Ampere fas 3, adr 3004*)
	
	_rU_L1_L2			:REAL;			(*Spänning L1-L2 i Volt, adr 3020*)
	_rU_L2_L3			:REAL;			(*Spänning L2-L3 i Volt, adr 3022*)
	_rU_L3_L1			:REAL;			(*Spänning L3-L1 i Volt, adr 3024*)
										
	_rU_L1_N			:REAL;			(*Spänning L1-N i Volt, adr 3028*)
	_rU_L2_N			:REAL;			(*Spänning L2-N i Volt, adr 3030*)
	_rU_L3_N			:REAL;			(*Spänning L3-N i Volt, adr 3032*)
										
	_rP1				:REAL;			(*Effekt fas 1 i kW, adr 3054*)
	_rP2				:REAL;			(*Effekt fas 2 i kW, adr 3056*)
	_rP3				:REAL;			(*Effekt fas 3 i kW, adr 3058*)									
	_rPtot				:REAL;			(*Total aktiv effekt i kW, adr 3060*)
	_rPVAR				:REAL;			(*Total reaktiv effekt i kVAR, adr 3068*)
	_rPVA				:REAL;			(*Total apparent effekt i kVA, adr 3076*)
										
	_rPfa				:REAL;			(*Effektfaktor , adr 3084*)
										
	_rHZ				:REAL;			(*Frekvens , adr 3110*)
										
	_rWHAI				:REAL;			(*Total aktiv energi import i Wh, adr 45100*)
	_rWHAE				:REAL;			(*Total aktiv energi export i Wh, adr 45102*)
	_rVARHI				:REAL;			(*Total reaktiv energi import i VARh, adr 45104*)
	_rVARHE				:REAL;			(*Total reaktiv energi export i VARh, adr 45106*)
																			
	_rWHPAI			:REAL;			(*Partial aktiv energi import i Wh, adr 45108*)
	_rWHPAE			:REAL;			(*Partial reaktiv energi import i Wh, adr 45110*)
										
	_rWHAEI1			:REAL;			(*Aktiv energi import i Wh fas 1, adr 45112*)
	_rWHAEI2			:REAL;			(*Aktiv energi import i Wh fas 2, adr 45114*)
	_rWHAEI3			:REAL;			(*Aktiv energi import i Wh fas 3, adr 45116*)
																			
	
END_VAR
VAR
	fbRtuMaster:		ModbusRtuMaster_KL6x22B; 		(*Modbus master instans*)
	fbDelay:			TON;							(*Fördröjning mellan sekvenserna*)
	nStat:					INT := 0;					(*Sekvens*)
	stIEM_Data:ST_IEM3255;	
END_VAR

CASE nStat OF

0:(*Start steg*)
	IF bEnable THEN
		bMbCommErr := FALSE;
		bBusy := TRUE;
		nStat := 2;
	END_IF


2:(*Modbus Funktion 3, Läs data från Holding Registers*)
fbRtuMaster.ReadRegs(
					UnitID:= bySlaveAdr ,
					Quantity:= 6,
					MBAddr:= 2998 ,
					cbLength:= SIZEOF(stIEM_Data.stCurrent) ,
					pMemoryAddr:=  ADR(stIEM_Data.stCurrent),
					Execute:= TRUE ,
					Timeout:= T#2s ,BUSY=> ,	Error=> , ErrorId=> ,cbRead=> );

IF fbRtuMaster.Error THEN
	nStat := 999;
ELSIF  NOT fbRtuMaster.BUSY AND NOT fbRtuMaster.Error THEN
	fbRtuMaster.ReadRegs(Execute := FALSE);
	nStat := 3;
END_IF


3:	(*Fördröj*)
fbDelay(IN:= TRUE, PT:=T#100ms , Q=> , ET=> );
IF fbDelay.Q THEN
	fbDelay(IN:= FALSE);
	nStat := 4;
END_IF;


4:(*Modbus Funktion 3, Läs data från Holding Registers*)
fbRtuMaster.ReadRegs(
					UnitID:= bySlaveAdr ,
					Quantity:= 6,
					MBAddr:= 3020 ,
					cbLength:= SIZEOF(stIEM_Data.stVolt) ,
					pMemoryAddr:=  ADR(stIEM_Data.stVolt),
					Execute:= TRUE ,
					Timeout:= T#2s ,BUSY=> ,	Error=> , ErrorId=> ,cbRead=> );

IF fbRtuMaster.Error THEN
	nStat := 999;
ELSIF  NOT fbRtuMaster.BUSY AND NOT fbRtuMaster.Error THEN
	fbRtuMaster.ReadRegs(Execute := FALSE);
	nStat := 5;
END_IF


5:	(*Fördröj*)
fbDelay(IN:= TRUE, PT:=T#100MS , Q=> , ET=> );
IF fbDelay.Q THEN
	fbDelay(IN:= FALSE);
	nStat := 6;
END_IF;

6:(*Modbus Funktion 3, Läs data från Holding Registers*)
fbRtuMaster.ReadRegs(
					UnitID:= bySlaveAdr ,
					Quantity:= 6,
					MBAddr:= 3028 ,
					cbLength:= SIZEOF(stIEM_Data.stVolt2) ,
					pMemoryAddr:=  ADR(stIEM_Data.stVolt2),
					Execute:= TRUE ,
					Timeout:= T#2s ,BUSY=> ,	Error=> , ErrorId=> ,cbRead=> );


					
IF fbRtuMaster.Error THEN
	nStat := 999;
ELSIF  NOT fbRtuMaster.BUSY AND NOT fbRtuMaster.Error THEN
	fbRtuMaster.ReadRegs(Execute := FALSE);
	nStat := 7;
END_IF


7:	(*Fördröj*)
fbDelay(IN:= TRUE, PT:=T#100MS , Q=> , ET=> );
IF fbDelay.Q THEN
	fbDelay(IN:= FALSE);
	nStat := 8;
END_IF;


8:(*Modbus Funktion 3, Läs data från Holding Registers*)
fbRtuMaster.ReadRegs(
					UnitID:= bySlaveAdr ,
					Quantity:= 8,
					MBAddr:= 3052 ,
					cbLength:= SIZEOF(stIEM_Data.stPower) ,
					pMemoryAddr:=  ADR(stIEM_Data.stPower),
					Execute:= TRUE ,
					Timeout:= T#2s ,BUSY=> ,	Error=> , ErrorId=> ,cbRead=> );

IF fbRtuMaster.Error THEN
	nStat := 999;
ELSIF  NOT fbRtuMaster.BUSY AND NOT fbRtuMaster.Error THEN
	fbRtuMaster.ReadRegs(Execute := FALSE);
	nStat := 9;
END_IF


9:	(*Fördröj*)
fbDelay(IN:= TRUE, PT:=T#100ms , Q=> , ET=> );
IF fbDelay.Q THEN
	fbDelay(IN:= FALSE);
	nStat := 10;
END_IF;

10:(*Modbus Funktion 3, Läs data från Holding Registers*)
fbRtuMaster.ReadRegs(
					UnitID:= bySlaveAdr ,
					Quantity:= 10,
					MBAddr:= 3066 ,
					cbLength:= SIZEOF(stIEM_Data.stPower2) ,
					pMemoryAddr:=  ADR(stIEM_Data.stPower2),
					Execute:= TRUE ,
					Timeout:= T#2s ,BUSY=> ,	Error=> , ErrorId=> ,cbRead=> );

IF fbRtuMaster.Error THEN
	nStat := 999;
ELSIF  NOT fbRtuMaster.BUSY AND NOT fbRtuMaster.Error THEN
	fbRtuMaster.ReadRegs(Execute := FALSE);
	nStat := 11;
END_IF


11:	(*Fördröj*)
fbDelay(IN:= TRUE, PT:=T#100ms , Q=> , ET=> );
IF fbDelay.Q THEN
	fbDelay(IN:= FALSE);
	nStat := 12;
END_IF;


12:(*Modbus Funktion 3, Läs data från Holding Registers*)
fbRtuMaster.ReadRegs(
					UnitID:= bySlaveAdr ,
					Quantity:= 2,
					MBAddr:= 3082 ,
					cbLength:= SIZEOF(stIEM_Data.stPowerFactor) ,
					pMemoryAddr:=  ADR(stIEM_Data.stPowerFactor),
					Execute:= TRUE ,
					Timeout:= T#2s ,BUSY=> ,	Error=> , ErrorId=> ,cbRead=> );

IF fbRtuMaster.Error THEN
	nStat := 999;
ELSIF  NOT fbRtuMaster.BUSY AND NOT fbRtuMaster.Error THEN
	fbRtuMaster.ReadRegs(Execute := FALSE);
	nStat := 13;
END_IF


13:	(*Fördröj*)
fbDelay(IN:= TRUE, PT:=T#100ms , Q=> , ET=> );
IF fbDelay.Q THEN
	fbDelay(IN:= FALSE);
	nStat := 14;
END_IF;

14:(*Modbus Funktion 3, Läs data från Holding Registers*)
fbRtuMaster.ReadRegs(
					UnitID:= bySlaveAdr ,
					Quantity:= 2,
					MBAddr:= 3108 ,
					cbLength:= SIZEOF(stIEM_Data.stFrequency) ,
					pMemoryAddr:=  ADR(stIEM_Data.stFrequency),
					Execute:= TRUE ,
					Timeout:= T#2s ,BUSY=> ,	Error=> , ErrorId=> ,cbRead=> );

IF fbRtuMaster.Error THEN
	nStat := 999;
ELSIF  NOT fbRtuMaster.BUSY AND NOT fbRtuMaster.Error THEN
	fbRtuMaster.ReadRegs(Execute := FALSE);
	nStat := 15;
END_IF


15:	(*Fördröj*)
fbDelay(IN:= TRUE, PT:=T#100ms , Q=> , ET=> );
IF fbDelay.Q THEN
	fbDelay(IN:= FALSE);
	nStat := 16;
END_IF;

16:(*Modbus Funktion 3, Läs data från Holding Registers*)
fbRtuMaster.ReadRegs(
					UnitID:= bySlaveAdr ,
					Quantity:= 8,
					MBAddr:= 45100 ,
					cbLength:= SIZEOF(stIEM_Data.stTotalEnergy) ,
					pMemoryAddr:=  ADR(stIEM_Data.stTotalEnergy),
					Execute:= TRUE ,
					Timeout:= T#2s ,BUSY=> ,	Error=> , ErrorId=> ,cbRead=> );

IF fbRtuMaster.Error THEN
	nStat := 999;
ELSIF  NOT fbRtuMaster.BUSY AND NOT fbRtuMaster.Error THEN
	fbRtuMaster.ReadRegs(Execute := FALSE);
	nStat := 17;
END_IF


17:	(*Fördröj*)
fbDelay(IN:= TRUE, PT:=T#100ms , Q=> , ET=> );
IF fbDelay.Q THEN
	fbDelay(IN:= FALSE);
	nStat := 18;
END_IF;

18:(*Modbus Funktion 3, Läs data från Holding Registers*)
fbRtuMaster.ReadRegs(
					UnitID:= bySlaveAdr ,
					Quantity:= 4,
					MBAddr:= 45108 ,
					cbLength:= SIZEOF(stIEM_Data.stPartialEnergy) ,
					pMemoryAddr:=  ADR(stIEM_Data.stPartialEnergy),
					Execute:= TRUE ,
					Timeout:= T#2s ,BUSY=> ,	Error=> , ErrorId=> ,cbRead=> );

IF fbRtuMaster.Error THEN
	nStat := 999;
ELSIF  NOT fbRtuMaster.BUSY AND NOT fbRtuMaster.Error THEN
	fbRtuMaster.ReadRegs(Execute := FALSE);
	nStat := 19;
END_IF


19:	(*Fördröj*)
fbDelay(IN:= TRUE, PT:=T#100ms , Q=> , ET=> );
IF fbDelay.Q THEN
	fbDelay(IN:= FALSE);
	nStat := 20;
END_IF;


20:	(*Fördröj*)
fbDelay(IN:= TRUE, PT:=T#100ms , Q=> , ET=> );
IF fbDelay.Q THEN
	fbDelay(IN:= FALSE);
	nStat := 21;
END_IF;

21:(*Modbus Funktion 3, Läs data från Holding Registers*)
fbRtuMaster.ReadRegs(
					UnitID:= bySlaveAdr ,
					Quantity:= 6,
					MBAddr:= 45110 ,
					cbLength:= SIZEOF(stIEM_Data.stPhaseEnergy) ,
					pMemoryAddr:=  ADR(stIEM_Data.stPhaseEnergy),
					Execute:= TRUE ,
					Timeout:= T#2s ,BUSY=> ,	Error=> , ErrorId=> ,cbRead=> );

IF fbRtuMaster.Error THEN
	nStat := 999;
ELSIF  NOT fbRtuMaster.BUSY AND NOT fbRtuMaster.Error THEN
	fbRtuMaster.ReadRegs(Execute := FALSE);
	nStat := 22;
END_IF


22:	(*Fördröj*)
fbDelay(IN:= TRUE, PT:=T#100ms , Q=> , ET=> );
IF fbDelay.Q THEN
	fbDelay(IN:= FALSE);
	nStat := 23;
END_IF;


23:(*Modbus Funktion 3, Läs data från Holding Registers*)
fbRtuMaster.ReadRegs(
					UnitID:= bySlaveAdr ,
					Quantity:= 2,
					MBAddr:= 45011 ,
					cbLength:= SIZEOF(stIEM_Data.stAlarmValue) ,
					pMemoryAddr:=  ADR(stIEM_Data.stAlarmValue),
					Execute:= TRUE ,
					Timeout:= T#2s ,BUSY=> ,	Error=> , ErrorId=> ,cbRead=> );

IF fbRtuMaster.Error THEN
	nStat := 999;
ELSIF  NOT fbRtuMaster.BUSY AND NOT fbRtuMaster.Error THEN
	fbRtuMaster.ReadRegs(Execute := FALSE);
	nStat := 24;
END_IF


24:	(*Fördröj*)
fbDelay(IN:= TRUE, PT:=T#100ms , Q=> , ET=> );
IF fbDelay.Q THEN
	fbDelay(IN:= FALSE);
	nStat := 40;
END_IF;

40:(*Läsning klar*)
	(*Beräkna och visa på utgången*)
	_rI1:= 		STIEM_Data.stCurrent.Phase_1_current;
	_rI2:=		STIEM_Data.stCurrent.Phase_2_current;
	_rI3:=		STIEM_Data.stCurrent.Phase_3_current;	
	_rU_L1_L2:=	STIEM_Data.stVolt.Voltage_L1_L2;
	_rU_L2_L3:=	STIEM_Data.stVolt.Voltage_L2_L3;
	_rU_L3_L1:=	STIEM_Data.stVolt.Voltage_L3_L1;	
	_rU_L1_N:=	STIEM_Data.stVolt2.Voltage_L1_N;
	_rU_L2_N:=	STIEM_Data.stVolt2.Voltage_L2_N;
	_rU_L3_N:=	STIEM_Data.stVolt2.Voltage_L3_N;
	_rP1:=		STIEM_Data.stPower.Active_Power_Phase_1;
	_rP2:=		STIEM_Data.stPower.Active_Power_Phase_2;
	_rP3:=		STIEM_Data.stPower.Active_Power_Phase_3;
	_rPtot:=	STIEM_Data.stPower.Total_Active_Power;
	_rPVAR:=	STIEM_Data.stPower2.Total_Reactive_Power;
	_rPVA:=		STIEM_Data.stPower2.Total_Apparent_Power;
	_rPfa:=		STIEM_Data.stPowerFactor.Total_Power_Factor;
	_rHZ:=		STIEM_Data.stFrequency.Frequency;
	_rWHAI:=	STIEM_Data.stTotalEnergy.Total_Active_Energy_Import;
	_rWHAE:=	STIEM_Data.stTotalEnergy.Total_Active_Energy_Export;
	_rVARHI:=	STIEM_Data.stTotalEnergy.Total_Reactive_Energy_Import;
	_rVARHE:=	STIEM_Data.stTotalEnergy.Total_Reactive_Energy_Export;
	_rWHPAI:=	STIEM_Data.stPartialEnergy.Partial_Active_Energy_Import;
	_rWHPAE:=	STIEM_Data.stPartialEnergy.Partial_Reactive_Energy_Import;
	_rWHAEI1:=	STIEM_Data.stPhaseEnergy.Active_Energy_Import_Phase_1;
	_rWHAEI2:=	STIEM_Data.stPhaseEnergy.Active_Energy_Import_Phase_2;
	_rWHAEI3:=	STIEM_Data.stPhaseEnergy.Active_Energy_Import_Phase_3;
	
	nStat := 0;

999:(*Något blev fel*)
	fbRtuMaster.ReadRegs(Execute := FALSE);
	bMbCommErr:= TRUE;
	bBusy := FALSE;
	nStat := 0;
END_CASE

END_FUNCTION_BLOCK

// ---- POUs/_FBs/FB_FL.TcPOU
FUNCTION_BLOCK FB_FL
VAR_INPUT
	Larm_in :BOOL;
	TID_in :INT;
END_VAR
VAR_OUTPUT
	Larm_ut :BOOL;
END_VAR
VAR
	TON_0: TON;
END_VAR

Larm_ut := TON_0.Q;
TON_0(IN := Larm_in, PT := INT_TO_TIME(TID_in) * 60000); // TON

END_FUNCTION_BLOCK

// ---- POUs/WXT530/F15_AS3_WXT530.TcPOU
PROGRAM F15_AS3_WXT530
VAR
	FB_WXT350_1: FB_WXT350;
	Enable:BOOL:=TRUE;
	FB_FL0: FB_FL;
	ComError :BOOL;
	
	TOF_0: TOF;
END_VAR


// PAGE
TOF_0(IN := FB_WXT350_1.ComError, PT := T#30s); // TOF
FB_WXT350_1(bEnable := GVL_Fastighet.WXT530); // FB_WXT350
GVL_WXT530._GW3U_DN := FB_WXT350_1._Dn;
ComError := NOT TOF_0.Q;
GVL_WXT530._GW3U_DM := FB_WXT350_1._Dm;
GVL_WXT530._GW3U_DX := FB_WXT350_1._Dx;
GVL_WXT530._GW3U_SN := FB_WXT350_1._Sn;
GVL_WXT530._GW3U_SM := FB_WXT350_1._Sm;
GVL_WXT530._GW3U_SX := FB_WXT350_1._Sx;
GVL_WXT530._GW3U_GT3U := FB_WXT350_1._Ta;
GVL_WXT530._GW3U_GT41 := FB_WXT350_1._TP;
GVL_WXT530._GW3U_GM41 := FB_WXT350_1._Ua;
GVL_WXT530._GW3U_GP41 := FB_WXT350_1._Pa;
GVL_WXT530._GW3U_RC := FB_WXT350_1._Rc;
GVL_WXT530._GW3U_RD := FB_WXT350_1._Rd;
GVL_WXT530._GW3U_RI := FB_WXT350_1._Ri;
GVL_WXT530._GW3U_HC := FB_WXT350_1._Hc;
GVL_WXT530._GW3U_HD := FB_WXT350_1._Hd;
GVL_WXT530._GW3U_HI := FB_WXT350_1._Hi;
GVL_WXT530._GW3U_RP := FB_WXT350_1._Rp;
GVL_WXT530._GW3U_HP := FB_WXT350_1._Hp;
FB_FL0(Larm_in := ComError, TID_in := GVL_Larm._GW3U_LC_FL); // FB_FL
GVL_Larm._GW3U_LC := FB_FL0.Larm_ut;

END_PROGRAM

// ---- POUs/_FBs/FB_WXT350.TcPOU
FUNCTION_BLOCK FB_WXT350

VAR_INPUT
	bEnable:BOOL;	
END_VAR

VAR
	fbSendString_Com1: SendString;
	fbReceiveString_Com1: ReceiveString;
	
	sReceivedCommand_Com1: STRING;
	sReceivedData_Com1: STRING;
	sLastCommand_Com1: STRING;
	
	sDeviceAdr 		:STRING:= '0';
	
	sSuffix : STRING:='$R$L';
	sPrefix1 : STRING;//:=CONCAT(sDeviceAdr, sCommand1);
	sPrefix2 : STRING;//:=CONCAT(sDeviceAdr, sCommand2);
	sPrefix3 : STRING;//:=CONCAT(sDeviceAdr, sCommand3);
	
	(*Wind Data Message (aR1)*)
	sCommand1 				:STRING:= 'R1';
	sReceivedString_Com1	:STRING(255); 	(* Dn=236D,Dm=283D,Dx=031D,Sn=0.0M,Sm=1.0M,Sx=2.2M *)
	sSendAdrCom1 			:STRING;	(*sDeviceAdr + sCommand1 = 0R1*)
	sSendCommand1			:STRING(255);
	
	(*Pressure, Temperature and Humidity Data Message (aR2)*)
	sCommand2 				:STRING:= 'R2';
	sReceivedString_Com2	:STRING(255);	(*0R2,Ta=23.6C,Ua=14.2P,Pa=1026.6H<cr><lf>*)
	sSendString2 			:STRING;
	sSendAdrCom2 			:STRING;	(*sDeviceAdr + sCommand2 = 0R2*)
	sSendCommand2			:STRING(255);
	
	(*Precipitation Data Message (aR3)*)
	sCommand3 				:STRING:= 'R3';
	sReceivedString_Com3	:STRING(255);	(*0R3,Rc=0.0M,Rd=0s,Ri=0.0M,Hc=0.0M,Hd=0s,Hi=0.0M,Rp=0.0M,Hp=0.0M<cr><lf>*)
	sSendString3 			:STRING;
	sSendAdrCom3 			:STRING;	(*sDeviceAdr + sCommand3 = 0R3*)
	sSendCommand3			:STRING(255);
	
	nState : INT; 
	nStateTON : TON;
	
	RunCounter: INT;


	
	
	
END_VAR

VAR_OUTPUT
	
	ComError	:BOOL;

(*Wind Data Message (aR1)*)
	_Dn	:REAL;  (*Wind direction minimum (D = degrees)*)
	_Dm	:REAL;  (*Wind direction average (D = degrees)*)
	_Dx	:REAL;  (*Wind direction maximum (D = degrees*)
	_Sn	:REAL;  (*Wind speed minimum (M = m/S)*)
	_Sm	:REAL;  (*Wind speed average (M = m/S)*)
	_Sx	:REAL;  (*Wind speed maximum (M = m/S)*)	
	
(*Pressure, Temperature and Humidity Data Message (aR2)*)
	_Ta	:REAL;  (*Air temperature (C = °C)*)
	_TP :REAL;	(*Internal temperature (C = °C)*)
	_Ua	:REAL;  (*Relative humidity (P = % RH)*)
	_Pa	:REAL;  (*Air pressure (H = hPa)*)
	
(*Precipitation Data Message (aR3)*)
	_Rc :REAL; (*Rain accumulation (M = mm)*)
	_Rd :REAL; (*Rain duration (S = S)*)
	_Ri :REAL;(*Rain intensity (M = mm/h)*)
	_Hc :REAL; (*Hail accumulation (M = hits/cm2)*)
	_Hd :REAL; (*Hail duration (S = S)*)
	_Hi :REAL; (*Hail intensity (M = hits/cm2h)*)
	_Rp :REAL; (*Rain peak intensity (M = mm/h)*)
	_Hp :REAL; (*Hail peak intensity (M = hits/cm2h)*)
	
	
	
END_VAR


ComError:= fbReceiveString_Com1.StringReceived;

CASE nState OF

	0: (* Init state *)
	IF bEnable THEN
		RunCounter:=RunCounter+1;
		nState := 10;
		END_IF	

	10: (* Send command:R1 *)	
		nStateTON(IN:=TRUE, PT:=T#200MS);
		
		sSendAdrCom1 := CONCAT(sDeviceAdr,sCommand1);
		sSendCommand1 := CONCAT(sSendAdrCom1,sSuffix);
		fbSendString_Com1(SendString:=sSendCommand1, TXbuffer:=GVL_WXT530.TxBuffer_Com1);
		
		sPrefix1 :=CONCAT(sDeviceAdr, sCommand1);
		
		IF nStateTON.Q THEN
			nStateTON(IN:=FALSE);
			nState := 20; //Change state
		END_IF
	
	20:	(* Wait for StringReceived command:R1 *)
		nStateTON(IN:=TRUE, PT:=T#5S);
	
		fbReceiveString_Com1(
			Prefix:=sPrefix1,
			Suffix:=sSuffix,
			Timeout:=T#500MS,
			Reset:= ,
			StringReceived=> ,
			Busy=> ,
			Error=> ,
			RxTimeout=> ,
			ReceivedString:=sReceivedString_Com1,
			RXbuffer:=GVL_WXT530.RxBuffer_Com1);
			
		IF fbReceiveString_Com1.StringReceived THEN
			nStateTON(IN:=FALSE);
			nState := 30;
		ELSIF nStateTON.Q THEN
			nStateTON(IN:=FALSE);
			nState := 40;
		END_IF
	
	30: (* Update values:R1 *)
		nStateTON(IN:=TRUE, PT:=T#200MS);
		
		_Dn	:= STRING_TO_REAL(MID(sReceivedString_Com1,6,FIND(sReceivedString_Com1,'Dn')+3));
		_Dm	:= STRING_TO_REAL(MID(sReceivedString_Com1,6,FIND(sReceivedString_Com1,'Dm')+3));
		_Dx	:= STRING_TO_REAL(MID(sReceivedString_Com1,6,FIND(sReceivedString_Com1,'Dx')+3));
		_Sn	:= STRING_TO_REAL(MID(sReceivedString_Com1,6,FIND(sReceivedString_Com1,'Sn')+3));
		_Sm	:= STRING_TO_REAL(MID(sReceivedString_Com1,6,FIND(sReceivedString_Com1,'Sm')+3));
		_Sx	:= STRING_TO_REAL(MID(sReceivedString_Com1,6,FIND(sReceivedString_Com1,'Sx')+3)); 
		
		IF nStateTON.Q THEN
			nStateTON(IN:=FALSE);
			nState := 40; //Change state
		END_IF
	
	40: (* Send command:R2 *)	
		nStateTON(IN:=TRUE, PT:=T#200MS);
		
		sSendAdrCom2 := CONCAT(sDeviceAdr,sCommand2);
		sSendCommand2 := CONCAT(sSendAdrCom2,sSuffix);
		fbSendString_Com1(SendString:=sSendCommand2, TXbuffer:=GVL_WXT530.TxBuffer_Com1);
		
		sPrefix2 := CONCAT(sDeviceAdr, sCommand2);
		
		IF nStateTON.Q THEN
			nStateTON(IN:=FALSE);
			nState := 50; //Change state
		END_IF
		
	50:	(* Wait for StringReceived command:R2 *)
		nStateTON(IN:=TRUE, PT:=T#5S);
		
		fbReceiveString_Com1(
			Prefix:=sPrefix2,
			Suffix:=sSuffix,
			Timeout:=T#500MS,
			Reset:= ,
			StringReceived=> ,
			Busy=> ,
			Error=> ,
			RxTimeout=> ,
			ReceivedString:=sReceivedString_Com2,
			RXbuffer:=GVL_WXT530.RxBuffer_Com1);
			
		IF fbReceiveString_Com1.StringReceived THEN
			nStateTON(IN:=FALSE);
			nState := 60;
		ELSIF nStateTON.Q THEN
			nStateTON(IN:=FALSE);
			nState := 70;
		END_IF
	
	60: (* Update values:R2 *)
		nStateTON(IN:=TRUE, PT:=T#200MS);
		
		(*Pressure, Temperature and Humidity Data Message (aR2)*)
		_Ta	:= STRING_TO_REAL(MID(sReceivedString_Com2,6,FIND(sReceivedString_Com2,'Ta')+3));
		_TP	:= STRING_TO_REAL(MID(sReceivedString_Com2,6,FIND(sReceivedString_Com2,'TP')+3));
		_Ua	:= STRING_TO_REAL(MID(sReceivedString_Com2,6,FIND(sReceivedString_Com2,'Ua')+3));
		_Pa	:= STRING_TO_REAL(MID(sReceivedString_Com2,6,FIND(sReceivedString_Com2,'Pa')+3)); 
		
		IF nStateTON.Q THEN
			nStateTON(IN:=FALSE);
			nState := 70; //Change state
		END_IF

70: (* Send command:R3 *)	
		nStateTON(IN:=TRUE, PT:=T#200MS);
		
		sSendAdrCom3 := CONCAT(sDeviceAdr,sCommand3);
		sSendCommand3 := CONCAT(sSendAdrCom3,sSuffix);
		fbSendString_Com1(SendString:=sSendCommand3, TXbuffer:=GVL_WXT530.TxBuffer_Com1);
		
		sPrefix3 := CONCAT(sDeviceAdr, sCommand3);
		
		IF nStateTON.Q THEN
			nStateTON(IN:=FALSE);
			nState := 80; //Change state
		END_IF
		
	80:	(* Wait for StringReceived command:R3 *)
		nStateTON(IN:=TRUE, PT:=T#5S);
		
		fbReceiveString_Com1(
			Prefix:=sPrefix3,
			Suffix:=sSuffix,
			Timeout:=T#500MS,
			Reset:= ,
			StringReceived=> ,
			Busy=> ,
			Error=> ,
			RxTimeout=> ,
			ReceivedString:=sReceivedString_Com3,
			RXbuffer:=GVL_WXT530.RxBuffer_Com1);
			
		IF fbReceiveString_Com1.StringReceived THEN
			nStateTON(IN:=FALSE);
			nState := 90;
		ELSIF nStateTON.Q THEN
			nStateTON(IN:=FALSE);
			nState := 90;
		END_IF
	
	90: (* Update values:R3 *)
		nStateTON(IN:=TRUE, PT:=T#200MS);
		
		_Rc	:= STRING_TO_REAL(MID(sReceivedString_Com3,6,FIND(sReceivedString_Com3,'Rc')+3));
		_Rd	:= STRING_TO_REAL(MID(sReceivedString_Com3,6,FIND(sReceivedString_Com3,'Rd')+3));
		_Ri	:= STRING_TO_REAL(MID(sReceivedString_Com3,6,FIND(sReceivedString_Com3,'Ri')+3));
		_Hc	:= STRING_TO_REAL(MID(sReceivedString_Com3,6,FIND(sReceivedString_Com3,'Hc')+3));
		_Hd	:= STRING_TO_REAL(MID(sReceivedString_Com3,6,FIND(sReceivedString_Com3,'Hd')+3));
		_Hi	:= STRING_TO_REAL(MID(sReceivedString_Com3,6,FIND(sReceivedString_Com3,'Hi')+3));
		_Rp	:= STRING_TO_REAL(MID(sReceivedString_Com3,6,FIND(sReceivedString_Com3,'Rp')+3));
		_Hp	:= STRING_TO_REAL(MID(sReceivedString_Com3,6,FIND(sReceivedString_Com3,'Hp')+3));
		
		IF nStateTON.Q THEN
			nStateTON(IN:=FALSE);
			nState := 0; //Change state
		END_IF
		



	

END_CASE

END_FUNCTION_BLOCK

// ---- POUs/WXT530/RS485.TcPOU
PROGRAM RS485
VAR
	fbSerialLineControl_Com1: SerialLineControl;
	ComIn_Com1 AT %I*: EL6inData22B;
	ComOut_Com1 AT %Q*:EL6outData22B;

	bRxData: BOOL;
	bTxData: BOOL;
END_VAR

fbSerialLineControl_Com1(
	Mode:=SERIALLINEMODE_EL6_22B,
	pComIn:=ADR(ComIn_Com1),
	pComOut:=ADR(ComOut_Com1),
	SizeComIn:=SIZEOF(ComIn_Com1),
	Error=> ,
	ErrorID=> ,
	TxBuffer:=GVL_WXT530.TxBuffer_Com1,
	RxBuffer:=GVL_WXT530.RxBuffer_Com1);

bRxData:=ComIn_Com1.D[0]<>0;
bTxData:=ComOut_Com1.D[0]<>0;

END_PROGRAM

// ---- POUs/MAIN.TcPOU
PROGRAM MAIN
VAR


END_VAR

(*Kalla på IOs*)
F15_AS3_AI();

(*Kalla på program*)

F15_ClusterCtrl();
F15_ClusterCtrl_Larm();


PLC_Batteri_Larm();
MAIN_loggning();

(*Kalla på Systemprogram*)
PersistentData();
PLC_TID();
WatchDog_PLC();

END_PROGRAM

// ---- POUs/IO/F15_AS3_AI.TcPOU
PROGRAM F15_AS3_AI
VAR
	
	AI_filter_0: AI_filter;
	AI_filter_1: AI_filter;
	AI_filter_2: AI_filter;
	AI_filter_3: AI_filter;
	AI_filter_4: AI_filter;
	AI_filter_5: AI_filter;
	AI_filter_6: AI_filter;
	AI_filter_7: AI_filter;

END_VAR

VAR PERSISTENT	
	
	Filtertid0 :INT;
	Filtertid1 :INT;
	Filtertid2 :INT;
	Filtertid3 :INT;
	Filtertid4 :INT;
	Filtertid5 :INT;
	Filtertid6 :INT;
	Filtertid7 :INT;
	
	Kalibrering0 :INT;
	Kalibrering1 :INT;
	Kalibrering2 :INT;
	Kalibrering3 :INT;
	Kalibrering4 :INT;
	Kalibrering5 :INT;
	Kalibrering6 :INT;
	Kalibrering7 :INT;
	
END_VAR


// PAGE
AI_filter_1(AI := GVL_IO._AI2, MVF := Kalibrering1, Filtertid := Filtertid1); // AI_filter
AI_filter_2(AI := GVL_IO._AI3, MVF := Kalibrering2, Filtertid := Filtertid2); // AI_filter
AI_filter_5(AI := GVL_IO._AI6, MVF := Kalibrering5, Filtertid := Filtertid5); // AI_filter
AI_filter_6(AI := GVL_IO._AI7, MVF := Kalibrering6, Filtertid := Filtertid6); // AI_filter
AI_filter_7(AI := GVL_IO._AI8, MVF := Kalibrering7, Filtertid := Filtertid7); // AI_filter
AI_filter_3(AI := GVL_IO._AI4, MVF := Kalibrering3, Filtertid := Filtertid3); // AI_filter
AI_filter_4(AI := GVL_IO._AI5, MVF := Kalibrering4, Filtertid := Filtertid4); // AI_filter
AI_filter_0(AI := GVL_IO._AI1, MVF := Kalibrering0, Filtertid := Filtertid0); // AI_filter
GVL_IO._GT41_MV := AI_filter_0.MV;
GVL_IO._GT42_MV := AI_filter_1.MV;
GVL_IO._GT43_MV := AI_filter_2.MV;
GVL_IO._GT44_MV := AI_filter_3.MV;
GVL_IO._GT45_MV := AI_filter_4.MV;
GVL_IO._GT46_MV := AI_filter_5.MV;
GVL_IO._GT47_MV := AI_filter_6.MV;
GVL_IO._GT48_MV := AI_filter_7.MV;

END_PROGRAM

// ---- POUs/_FBs/AI_filter.TcPOU
FUNCTION_BLOCK AI_filter
VAR_INPUT
	AI 				:INT;
	MVF				:INT;
	Filtertid 		:INT;
	
END_VAR
VAR_OUTPUT
	MV				:INT;
END_VAR
VAR
	Filter1			: FB_BA_FltrPT1;
END_VAR
VAR // added by the converter: edge detectors and wires of the graphical bodies
    _w1, _w2 : ANY;
END_VAR


// PAGE
Filter1(lrIn := AI, udiDampConst := _w1, bSetActl := FALSE); // FB_BA_FltrPT1
MV := _w2 + MVF;
_w1 := INT_TO_UDINT(Filtertid);
_w2 := LREAL_TO_INT(Filter1.lrOut);

END_FUNCTION_BLOCK

// ---- POUs/ClusterCtrl/F15_ClusterCtrl.TcPOU
PROGRAM F15_ClusterCtrl

VAR
	DeviceStatus1 :DWORD;
	DeviceStatus2 :DWORD;
	DeviceStatus3 :DWORD;
	
	
END_VAR

ClusterControl_3Unit();

GVL_ClusterCtrl._CCtrl_V1_P:= 				(F_WordSwap(ClusterControl_3Unit.stClusterCtrlData.stActivePower.ActivePower_Total))*0.001;
GVL_ClusterCtrl._CCtrl_V1_P1:= 				F_WordSwap(ClusterControl_3Unit.stClusterCtrlData.stActivePower.ActivePower_L1);	
GVL_ClusterCtrl._CCtrl_V1_P2:= 				F_WordSwap(ClusterControl_3Unit.stClusterCtrlData.stActivePower.ActivePower_L2);
GVL_ClusterCtrl._CCtrl_V1_P3:= 				F_WordSwap(ClusterControl_3Unit.stClusterCtrlData.stActivePower.ActivePower_L3);
GVL_ClusterCtrl._CCtrl_V1_U1_L1_N:=			(F_WordSwap(ClusterControl_3Unit.stClusterCtrlData.stLineVoltage.LineVoltage_L1_N)) /100; 	//Scaled to Volt
GVL_ClusterCtrl._CCtrl_V1_U2_L2_N:=			(F_WordSwap(ClusterControl_3Unit.stClusterCtrlData.stLineVoltage.LineVoltage_L2_N)) /100;	//Scaled to Volt
GVL_ClusterCtrl._CCtrl_V1_U3_L3_N:=			(F_WordSwap(ClusterControl_3Unit.stClusterCtrlData.stLineVoltage.LineVoltage_L3_N)) /100;	//Scaled to Volt
GVL_ClusterCtrl._CCtrl_V1_U1_L1_L2:=		F_WordSwap(ClusterControl_3Unit.stClusterCtrlData.stLineVoltage.LineVoltage_L1_L2);		
GVL_ClusterCtrl._CCtrl_V1_U2_L2_L3:=		F_WordSwap(ClusterControl_3Unit.stClusterCtrlData.stLineVoltage.LineVoltage_L1_L2);		
GVL_ClusterCtrl._CCtrl_V1_U3_L3_L1:=		F_WordSwap(ClusterControl_3Unit.stClusterCtrlData.stLineVoltage.LineVoltage_L3_L1);	
GVL_ClusterCtrl._CCtrl_V1_Itot:=			F_WordSwap(ClusterControl_3Unit.stClusterCtrlData.stLineCurrent.LineCurrent_Total);	
GVL_ClusterCtrl._CCtrl_V1_I1:=				(F_WordSwap(ClusterControl_3Unit.stClusterCtrlData.stLineCurrent.LineCurrent_L1)) / 1000; 	// Scaled to Ampere	
GVL_ClusterCtrl._CCtrl_V1_I2:=				(F_WordSwap(ClusterControl_3Unit.stClusterCtrlData.stLineCurrent.LineCurrent_L2)) / 1000;	// Scaled to Ampere	
GVL_ClusterCtrl._CCtrl_V1_I3:=				(F_WordSwap(ClusterControl_3Unit.stClusterCtrlData.stLineCurrent.LineCurrent_L3)) / 1000;	// Scaled to Ampere	
//GVL_ClusterCtrl._CCtrl_V1_Yield_Wh:=		F_WordSwap(ClusterControl_3Unit.stClusterCtrlData.stYield.Total_AC_energy_all_conductors_Wh);		
GVL_ClusterCtrl._CCtrl_V1_Yield_KWh:=		F_WordSwap(ClusterControl_3Unit.stClusterCtrlData.stYield.Total_AC_energy_all_conductors_kWh);		
GVL_ClusterCtrl._CCtrl_V1_Yield_MWh:=		F_WordSwap(ClusterControl_3Unit.stClusterCtrlData.stYield.Total_AC_energy_all_conductors_MWh);		
//GVL_ClusterCtrl._CCtrl_V1_YieldDay_Wh:=	F_WordSwap(ClusterControl_3Unit.stClusterCtrlData.stYield.Energy_current_day_all_conductors_Wh);		
GVL_ClusterCtrl._CCtrl_V1_YieldDay_kWh:=	F_WordSwap(ClusterControl_3Unit.stClusterCtrlData.stYield.Energy_current_day_all_conductors_kWh);		
GVL_ClusterCtrl._CCtrl_V1_PV:=				F_WordSwap(ClusterControl_3Unit.stClusterCtrlData.stPVDATA.PV_Power);	
GVL_ClusterCtrl._CCtrl_V1_HZ:=				(F_WordSwap(ClusterControl_3Unit.stClusterCtrlData.stLineCurrent.PowerFrequency)) / 100; //Scaled to Hz
GVL_ClusterCtrl._CCtrl_V1_APtot:=			F_WordSwap(ClusterControl_3Unit.stClusterCtrlData.stApparentPower.ApparentPower_Total);
GVL_ClusterCtrl._CCtrl_V1_AP1:=				F_WordSwap(ClusterControl_3Unit.stClusterCtrlData.stApparentPower.ApparentPower_L1);
GVL_ClusterCtrl._CCtrl_V1_AP2:=				F_WordSwap(ClusterControl_3Unit.stClusterCtrlData.stApparentPower.ApparentPower_L2);
GVL_ClusterCtrl._CCtrl_V1_AP3:=				F_WordSwap(ClusterControl_3Unit.stClusterCtrlData.stApparentPower.ApparentPower_L3);
GVL_ClusterCtrl._CCtrl_V1_RPtot:=			F_WordSwap(ClusterControl_3Unit.stClusterCtrlData.stReactivePower.ReactivePower_Total);
GVL_ClusterCtrl._CCtrl_V1_RP1:=				F_WordSwap(ClusterControl_3Unit.stClusterCtrlData.stReactivePower.ReactivePower_L1);
GVL_ClusterCtrl._CCtrl_V1_RP2:=				F_WordSwap(ClusterControl_3Unit.stClusterCtrlData.stReactivePower.ReactivePower_L2);
GVL_ClusterCtrl._CCtrl_V1_RP3:=				F_WordSwap(ClusterControl_3Unit.stClusterCtrlData.stReactivePower.ReactivePower_L3);
GVL_ClusterCtrl._CCtrl_V1_EnSaveMode:=		F_WordSwap(ClusterControl_3Unit.stClusterCtrlData.nEnergySavingMode);
GVL_ClusterCtrl._CCtrl_V1_TECInt:=			F_WordSwap(ClusterControl_3Unit.stClusterCtrlData.nTotEnergyConsInternally);
DeviceStatus1:=								F_WordSwap(ClusterControl_3Unit.stClusterCtrlData.stStatus.Device_Status);

GVL_ClusterCtrl._CCtrl_V2_P:= 				(F_WordSwap(ClusterControl_3Unit.stClusterCtrlData2.stActivePower.ActivePower_Total))*0.001;			
GVL_ClusterCtrl._CCtrl_V2_P1:= 				F_WordSwap(ClusterControl_3Unit.stClusterCtrlData2.stActivePower.ActivePower_L1);			
GVL_ClusterCtrl._CCtrl_V2_P2:= 				F_WordSwap(ClusterControl_3Unit.stClusterCtrlData2.stActivePower.ActivePower_L2);			
GVL_ClusterCtrl._CCtrl_V2_P3:= 				F_WordSwap(ClusterControl_3Unit.stClusterCtrlData2.stActivePower.ActivePower_L3);			
GVL_ClusterCtrl._CCtrl_V2_U1_L1_N:=			(F_WordSwap(ClusterControl_3Unit.stClusterCtrlData2.stLineVoltage.LineVoltage_L1_N)) / 100;	//Scaled to Volt			
GVL_ClusterCtrl._CCtrl_V2_U2_L2_N:=			(F_WordSwap(ClusterControl_3Unit.stClusterCtrlData2.stLineVoltage.LineVoltage_L2_N)) / 100;	//Scaled to Volt			
GVL_ClusterCtrl._CCtrl_V2_U3_L3_N:=			(F_WordSwap(ClusterControl_3Unit.stClusterCtrlData2.stLineVoltage.LineVoltage_L3_N)) / 100;	//Scaled to Volt			
GVL_ClusterCtrl._CCtrl_V2_U1_L1_L2:=		F_WordSwap(ClusterControl_3Unit.stClusterCtrlData2.stLineVoltage.LineVoltage_L1_L2);					
GVL_ClusterCtrl._CCtrl_V2_U2_L2_L3:=		F_WordSwap(ClusterControl_3Unit.stClusterCtrlData2.stLineVoltage.LineVoltage_L1_L2);					
GVL_ClusterCtrl._CCtrl_V2_U3_L3_L1:=		F_WordSwap(ClusterControl_3Unit.stClusterCtrlData2.stLineVoltage.LineVoltage_L3_L1);
GVL_ClusterCtrl._CCtrl_V2_Itot:=			F_WordSwap(ClusterControl_3Unit.stClusterCtrlData2.stLineCurrent.LineCurrent_Total);						
GVL_ClusterCtrl._CCtrl_V2_I1:=				(F_WordSwap(ClusterControl_3Unit.stClusterCtrlData2.stLineCurrent.LineCurrent_L1)) / 1000; 	// Scaled to Ampere					
GVL_ClusterCtrl._CCtrl_V2_I2:=				(F_WordSwap(ClusterControl_3Unit.stClusterCtrlData2.stLineCurrent.LineCurrent_L2)) / 1000;	// Scaled to Ampere 					
GVL_ClusterCtrl._CCtrl_V2_I3:=				(F_WordSwap(ClusterControl_3Unit.stClusterCtrlData2.stLineCurrent.LineCurrent_L3)) / 1000;	// Scaled to Ampere 					
//GVL_ClusterCtrl._CCtrl_V2_Yield_Wh:=		F_WordSwap(ClusterControl_3Unit.stClusterCtrlData2.stYield.Total_AC_energy_all_conductors_Wh);					
GVL_ClusterCtrl._CCtrl_V2_Yield_KWh:=		F_WordSwap(ClusterControl_3Unit.stClusterCtrlData2.stYield.Total_AC_energy_all_conductors_kWh);					
GVL_ClusterCtrl._CCtrl_V2_Yield_MWh:=		F_WordSwap(ClusterControl_3Unit.stClusterCtrlData2.stYield.Total_AC_energy_all_conductors_MWh);					
//GVL_ClusterCtrl._CCtrl_V2_YieldDay_Wh:=		F_WordSwap(ClusterControl_3Unit.stClusterCtrlData2.stYield.Energy_current_day_all_conductors_Wh);					
GVL_ClusterCtrl._CCtrl_V2_YieldDay_kWh:=	F_WordSwap(ClusterControl_3Unit.stClusterCtrlData2.stYield.Energy_current_day_all_conductors_kWh);					
GVL_ClusterCtrl._CCtrl_V2_PV:=				F_WordSwap(ClusterControl_3Unit.stClusterCtrlData2.stPVDATA.PV_Power);					
GVL_ClusterCtrl._CCtrl_V2_HZ:=				(F_WordSwap(ClusterControl_3Unit.stClusterCtrlData2.stLineCurrent.PowerFrequency)) / 100; //Scaled to Hz
GVL_ClusterCtrl._CCtrl_V2_APtot:=			F_WordSwap(ClusterControl_3Unit.stClusterCtrlData2.stApparentPower.ApparentPower_Total);
GVL_ClusterCtrl._CCtrl_V2_AP1:=				F_WordSwap(ClusterControl_3Unit.stClusterCtrlData2.stApparentPower.ApparentPower_L1);
GVL_ClusterCtrl._CCtrl_V2_AP2:=				F_WordSwap(ClusterControl_3Unit.stClusterCtrlData2.stApparentPower.ApparentPower_L2);
GVL_ClusterCtrl._CCtrl_V2_AP3:=				F_WordSwap(ClusterControl_3Unit.stClusterCtrlData2.stApparentPower.ApparentPower_L3);
GVL_ClusterCtrl._CCtrl_V2_RPtot:=			F_WordSwap(ClusterControl_3Unit.stClusterCtrlData2.stReactivePower.ReactivePower_Total);
GVL_ClusterCtrl._CCtrl_V2_RP1:=				F_WordSwap(ClusterControl_3Unit.stClusterCtrlData2.stReactivePower.ReactivePower_L1);
GVL_ClusterCtrl._CCtrl_V2_RP2:=				F_WordSwap(ClusterControl_3Unit.stClusterCtrlData2.stReactivePower.ReactivePower_L2);
GVL_ClusterCtrl._CCtrl_V2_RP3:=				F_WordSwap(ClusterControl_3Unit.stClusterCtrlData2.stReactivePower.ReactivePower_L3);
GVL_ClusterCtrl._CCtrl_V2_EnSaveMode:=		F_WordSwap(ClusterControl_3Unit.stClusterCtrlData2.nEnergySavingMode);
GVL_ClusterCtrl._CCtrl_V2_TECInt:=			F_WordSwap(ClusterControl_3Unit.stClusterCtrlData2.nTotEnergyConsInternally);
DeviceStatus2:=								F_WordSwap(ClusterControl_3Unit.stClusterCtrlData2.stStatus.Device_Status);					

GVL_ClusterCtrl._CCtrl_V3_P:= 				(F_WordSwap(ClusterControl_3Unit.stClusterCtrlData3.stActivePower.ActivePower_Total))*0.001;			
GVL_ClusterCtrl._CCtrl_V3_P1:= 				F_WordSwap(ClusterControl_3Unit.stClusterCtrlData3.stActivePower.ActivePower_L1);			
GVL_ClusterCtrl._CCtrl_V3_P2:= 				F_WordSwap(ClusterControl_3Unit.stClusterCtrlData3.stActivePower.ActivePower_L2);			
GVL_ClusterCtrl._CCtrl_V3_P3:= 				F_WordSwap(ClusterControl_3Unit.stClusterCtrlData3.stActivePower.ActivePower_L3);			
GVL_ClusterCtrl._CCtrl_V3_U1_L1_N:=			(F_WordSwap(ClusterControl_3Unit.stClusterCtrlData3.stLineVoltage.LineVoltage_L1_N)) / 100;	//Scaled to Volt				
GVL_ClusterCtrl._CCtrl_V3_U2_L2_N:=			(F_WordSwap(ClusterControl_3Unit.stClusterCtrlData3.stLineVoltage.LineVoltage_L2_N)) / 100;	//Scaled to Volt				
GVL_ClusterCtrl._CCtrl_V3_U3_L3_N:=			(F_WordSwap(ClusterControl_3Unit.stClusterCtrlData3.stLineVoltage.LineVoltage_L3_N)) / 100;	//Scaled to Volt				
GVL_ClusterCtrl._CCtrl_V3_U1_L1_L2:=		F_WordSwap(ClusterControl_3Unit.stClusterCtrlData3.stLineVoltage.LineVoltage_L1_L2);					
GVL_ClusterCtrl._CCtrl_V3_U2_L2_L3:=		F_WordSwap(ClusterControl_3Unit.stClusterCtrlData3.stLineVoltage.LineVoltage_L1_L2);					
GVL_ClusterCtrl._CCtrl_V3_U3_L3_L1:=		F_WordSwap(ClusterControl_3Unit.stClusterCtrlData3.stLineVoltage.LineVoltage_L3_L1);
GVL_ClusterCtrl._CCtrl_V3_Itot:=			F_WordSwap(ClusterControl_3Unit.stClusterCtrlData3.stLineCurrent.LineCurrent_Total);						
GVL_ClusterCtrl._CCtrl_V3_I1:=				(F_WordSwap(ClusterControl_3Unit.stClusterCtrlData3.stLineCurrent.LineCurrent_L1)) / 1000; 	// Scaled to Ampere					
GVL_ClusterCtrl._CCtrl_V3_I2:=				(F_WordSwap(ClusterControl_3Unit.stClusterCtrlData3.stLineCurrent.LineCurrent_L2)) / 1000;	// Scaled to Ampere 					
GVL_ClusterCtrl._CCtrl_V3_I3:=				(F_WordSwap(ClusterControl_3Unit.stClusterCtrlData3.stLineCurrent.LineCurrent_L3)) / 1000;	// Scaled to Ampere 					
//GVL_ClusterCtrl._CCtrl_V3_Yield_Wh:=		F_WordSwap(ClusterControl_3Unit.stClusterCtrlData3.stYield.Total_AC_energy_all_conductors_Wh);					
GVL_ClusterCtrl._CCtrl_V3_Yield_KWh:=		F_WordSwap(ClusterControl_3Unit.stClusterCtrlData3.stYield.Total_AC_energy_all_conductors_kWh);					
GVL_ClusterCtrl._CCtrl_V3_Yield_MWh:=		F_WordSwap(ClusterControl_3Unit.stClusterCtrlData3.stYield.Total_AC_energy_all_conductors_MWh);					
//GVL_ClusterCtrl._CCtrl_V3_YieldDay_Wh:=		F_WordSwap(ClusterControl_3Unit.stClusterCtrlData3.stYield.Energy_current_day_all_conductors_Wh);					
GVL_ClusterCtrl._CCtrl_V3_YieldDay_kWh:=	F_WordSwap(ClusterControl_3Unit.stClusterCtrlData3.stYield.Energy_current_day_all_conductors_kWh);					
GVL_ClusterCtrl._CCtrl_V3_PV:=				F_WordSwap(ClusterControl_3Unit.stClusterCtrlData3.stPVDATA.PV_Power);					
GVL_ClusterCtrl._CCtrl_V3_HZ:=				(F_WordSwap(ClusterControl_3Unit.stClusterCtrlData3.stLineCurrent.PowerFrequency)) / 100; //Scaled to Hz
GVL_ClusterCtrl._CCtrl_V3_APtot:=			F_WordSwap(ClusterControl_3Unit.stClusterCtrlData3.stApparentPower.ApparentPower_Total);
GVL_ClusterCtrl._CCtrl_V3_AP1:=				F_WordSwap(ClusterControl_3Unit.stClusterCtrlData3.stApparentPower.ApparentPower_L1);
GVL_ClusterCtrl._CCtrl_V3_AP2:=				F_WordSwap(ClusterControl_3Unit.stClusterCtrlData3.stApparentPower.ApparentPower_L2);
GVL_ClusterCtrl._CCtrl_V3_AP3:=				F_WordSwap(ClusterControl_3Unit.stClusterCtrlData3.stApparentPower.ApparentPower_L3);
GVL_ClusterCtrl._CCtrl_V3_RPtot:=			F_WordSwap(ClusterControl_3Unit.stClusterCtrlData3.stReactivePower.ReactivePower_Total);
GVL_ClusterCtrl._CCtrl_V3_RP1:=				F_WordSwap(ClusterControl_3Unit.stClusterCtrlData3.stReactivePower.ReactivePower_L1);
GVL_ClusterCtrl._CCtrl_V3_RP2:=				F_WordSwap(ClusterControl_3Unit.stClusterCtrlData3.stReactivePower.ReactivePower_L2);
GVL_ClusterCtrl._CCtrl_V3_RP3:=				F_WordSwap(ClusterControl_3Unit.stClusterCtrlData3.stReactivePower.ReactivePower_L3);
GVL_ClusterCtrl._CCtrl_V3_EnSaveMode:=		F_WordSwap(ClusterControl_3Unit.stClusterCtrlData3.nEnergySavingMode);
GVL_ClusterCtrl._CCtrl_V3_TECInt:=			F_WordSwap(ClusterControl_3Unit.stClusterCtrlData3.nTotEnergyConsInternally);
DeviceStatus3:=								F_WordSwap(ClusterControl_3Unit.stClusterCtrlData3.stStatus.Device_Status);

END_PROGRAM

// ---- POUs/_FBs/ClusterControl_3Unit.TcPOU
PROGRAM ClusterControl_3Unit
VAR_OUTPUT
	bBusy:					BOOL;		(*Upptagen med arbete*)
	bCommErr:				BOOL;		(*Modbus Kommunikationsfel*)												
END_VAR
VAR
	fbReadRegs:		FB_MBReadRegs; 						(*Modbus läs Holding Registers*)
	fbDelay:			TON;							(*Fördröjning mellan sekvenserna*)
	nStat:				INT := 0;						(*Sekvens*)
	bEnable			:BOOL:=TRUE;
	sSlaveIP 		:STRING:= '192.168.1.20';
	uiPort			:UINT:=502;	
	nUnit_ID				:BYTE:=4;
	nUnit_ID2				:BYTE:=5;	
	nUnit_ID3				:BYTE:=3;
	stClusterCtrlData: ST_ClusterCtrl;
	stClusterCtrlData2: ST_ClusterCtrl;
	stClusterCtrlData3: ST_ClusterCtrl;
	stClusterCtrlDataSensor:ST_ClusterCtrl;
END_VAR


CASE nStat OF

0:(*Start steg*)
	IF bEnable THEN
		bCommErr := FALSE;
		bBusy := TRUE;
		nStat := 2;
	END_IF

2:(*Modbus Funktion 3, Läs data från Holding Registers*)
fbReadRegs(
					sIPAddr:= sSlaveIP,
					nTCPPort:= uiPort,
					nUnitID:= nUnit_ID,
					nQuantity:= 8,
					nMBAddr:= 30775 ,
					cbLength:= SIZEOF(stClusterCtrlData.stActivePower) ,
					pDestAddr :=  ADR(stClusterCtrlData.stActivePower),
					bExecute:= TRUE ,
					tTimeout:= T#2S ,bBusy=> ,	bError=> , nErrId=> ,cbRead=> );
					

IF fbReadRegs.bError THEN
	nStat := 999;
ELSIF  NOT fbReadRegs.bBusy AND NOT fbReadRegs.bError THEN
	fbReadRegs(bExecute := FALSE);
	nStat := 3;
END_IF


3:	(*Fördröj*)
fbDelay(IN:= TRUE, PT:=T#200MS , Q=> , ET=> );
IF fbDelay.Q THEN
	fbDelay(IN:= FALSE);
	nStat := 4;
END_IF;


4:(*Modbus Funktion 3, Läs data från Holding Registers*)
fbReadRegs(
					sIPAddr:= sSlaveIP,
					nTCPPort:= uiPort,
					nUnitID:= nUnit_ID,
					nQuantity:= 12,
					nMBAddr:= 30783 ,
					cbLength:= SIZEOF(stClusterCtrlData.stLineVoltage) ,
					pDestAddr :=  ADR(stClusterCtrlData.stLineVoltage),
					bExecute:= TRUE ,
					tTimeout:= T#2S ,bBusy=> ,	bError=> , nErrId=> ,cbRead=> );
					

IF fbReadRegs.bError THEN
	nStat := 999;
ELSIF  NOT fbReadRegs.bBusy AND NOT fbReadRegs.bError THEN
	fbReadRegs(bExecute := FALSE);
	nStat := 5;
END_IF


5:	(*Fördröj*)
fbDelay(IN:= TRUE, PT:=T#200MS , Q=> , ET=> );
IF fbDelay.Q THEN
	fbDelay(IN:= FALSE);
	nStat := 6;
END_IF;


6:(*Modbus Funktion 3, Läs data från Holding Registers*)
(*Detta är den som fixar modbus *)
fbReadRegs(
					sIPAddr:= sSlaveIP,
					nTCPPort:= uiPort,
					nUnitID:= nUnit_ID,
					nQuantity:= 10,
					nMBAddr:= 30795 ,
					cbLength:= SIZEOF(stClusterCtrlData.stLineCurrent) ,
					pDestAddr :=  ADR(stClusterCtrlData.stLineCurrent),
					bExecute:= TRUE ,
					tTimeout:= T#2S ,bBusy=> ,	bError=> , nErrId=> ,cbRead=> );
					

IF fbReadRegs.bError THEN
	nStat := 999;
ELSIF  NOT fbReadRegs.bBusy AND NOT fbReadRegs.bError THEN
	fbReadRegs(bExecute := FALSE);
	nStat := 7;
END_IF


7:	(*Fördröj*)
fbDelay(IN:= TRUE, PT:=T#200MS , Q=> , ET=> );
IF fbDelay.Q THEN
	fbDelay(IN:= FALSE);
	nStat := 8;
END_IF;


8:(*Modbus Funktion 3, Läs data från Holding Registers*)
fbReadRegs(
					sIPAddr:= sSlaveIP,
					nTCPPort:= uiPort,
					nUnitID:= nUnit_ID,
					nQuantity:= 16,
					nMBAddr:= 30529 ,
					cbLength:= SIZEOF(stClusterCtrlData.stYield) ,
					pDestAddr :=  ADR(stClusterCtrlData.stYield),
					bExecute:= TRUE ,
					tTimeout:= T#2S ,bBusy=> ,	bError=> , nErrId=> ,cbRead=> );
					

IF fbReadRegs.bError THEN
	nStat := 999;
ELSIF  NOT fbReadRegs.bBusy AND NOT fbReadRegs.bError THEN
	fbReadRegs(bExecute := FALSE);
	nStat := 9;
END_IF


9:	(*Fördröj*)
fbDelay(IN:= TRUE, PT:=T#200MS , Q=> , ET=> );
IF fbDelay.Q THEN
	fbDelay(IN:= FALSE);
	nStat := 10;
END_IF;


10:(*Modbus Funktion 3, Läs data från Holding Registers*)
fbReadRegs(
					sIPAddr:= sSlaveIP,
					nTCPPort:= uiPort,
					nUnitID:= nUnit_ID,
					nQuantity:= 8,
					nMBAddr:= 30977 ,
					cbLength:= SIZEOF(stClusterCtrlData.stPVDATA) ,
					pDestAddr :=  ADR(stClusterCtrlData.stPVDATA),
					bExecute:= TRUE ,
					tTimeout:= T#2S ,bBusy=> ,	bError=> , nErrId=> ,cbRead=> );
					

IF fbReadRegs.bError THEN
	nStat := 999;
ELSIF  NOT fbReadRegs.bBusy AND NOT fbReadRegs.bError THEN
	fbReadRegs(bExecute := FALSE);
	nStat := 11;
END_IF


11:	(*Fördröj*)
fbDelay(IN:= TRUE, PT:=T#200MS , Q=> , ET=> );
IF fbDelay.Q THEN
	fbDelay(IN:= FALSE);
	nStat := 12;
END_IF;

12:(*Modbus Funktion 3, Läs data från Holding Registers*)
fbReadRegs(
					sIPAddr:= sSlaveIP,
					nTCPPort:= uiPort,
					nUnitID:= nUnit_ID,
					nQuantity:= 2,
					nMBAddr:= 30201 ,
					cbLength:= SIZEOF(stClusterCtrlData.stStatus) ,
					pDestAddr :=  ADR(stClusterCtrlData.stStatus),
					bExecute:= TRUE ,
					tTimeout:= T#2S ,bBusy=> ,	bError=> , nErrId=> ,cbRead=> );
					

IF fbReadRegs.bError THEN
	nStat := 999;
ELSIF  NOT fbReadRegs.bBusy AND NOT fbReadRegs.bError THEN
	fbReadRegs(bExecute := FALSE);
	nStat := 13;
END_IF


13:	(*Fördröj*)
fbDelay(IN:= TRUE, PT:=T#200MS , Q=> , ET=> );
IF fbDelay.Q THEN
	fbDelay(IN:= FALSE);
	nStat := 14;
END_IF;

14: (* nTotEnergyConsInternally *) 
fbReadRegs(
					sIPAddr:= sSlaveIP,
					nTCPPort:= uiPort,
					nUnitID:= nUnit_ID,
					nQuantity:= 2,
					nMBAddr:= 30593 ,
					cbLength:= SIZEOF(stClusterCtrlData.nTotEnergyConsInternally) ,
					pDestAddr :=  ADR(stClusterCtrlData.nTotEnergyConsInternally),
					bExecute:= TRUE ,
					tTimeout:= T#2S ,bBusy=> ,	bError=> , nErrId=> ,cbRead=> );
					

IF fbReadRegs.bError THEN
	nStat := 999;
ELSIF  NOT fbReadRegs.bBusy AND NOT fbReadRegs.bError THEN
	fbReadRegs(bExecute := FALSE);
	nStat := 15;
END_IF

15:	(*Fördröj*)
fbDelay(IN:= TRUE, PT:=T#200MS , Q=> , ET=> );
IF fbDelay.Q THEN
	fbDelay(IN:= FALSE);
	nStat := 16;
END_IF;

16: (* nInverterInteriorTemp *) 
fbReadRegs(
					sIPAddr:= sSlaveIP,
					nTCPPort:= uiPort,
					nUnitID:= nUnit_ID,
					nQuantity:= 2,
					nMBAddr:= 34113 ,
					cbLength:= SIZEOF(stClusterCtrlData.nInverterInteriorTemp) ,
					pDestAddr :=  ADR(stClusterCtrlData.nInverterInteriorTemp),
					bExecute:= TRUE ,
					tTimeout:= T#2S ,bBusy=> ,	bError=> , nErrId=> ,cbRead=> );
					

IF fbReadRegs.bError THEN
	nStat := 999;
ELSIF  NOT fbReadRegs.bBusy AND NOT fbReadRegs.bError THEN
	fbReadRegs(bExecute := FALSE);
	nStat := 17;
END_IF

17:	(*Fördröj*)
fbDelay(IN:= TRUE, PT:=T#200MS , Q=> , ET=> );
IF fbDelay.Q THEN
	fbDelay(IN:= FALSE);
	nStat := 18;
END_IF;	

18:(*ReactivePower*)
fbReadRegs(
					sIPAddr:= sSlaveIP,
					nTCPPort:= uiPort,
					nUnitID:= nUnit_ID,
					nQuantity:= 8,
					nMBAddr:= 30805 ,
					cbLength:= SIZEOF(stClusterCtrlData.stReactivePower) ,
					pDestAddr :=  ADR(stClusterCtrlData.stReactivePower),
					bExecute:= TRUE ,
					tTimeout:= T#2S ,bBusy=> ,	bError=> , nErrId=> ,cbRead=> );
					

IF fbReadRegs.bError THEN
	nStat := 999;
ELSIF  NOT fbReadRegs.bBusy AND NOT fbReadRegs.bError THEN
	fbReadRegs(bExecute := FALSE);
	nStat := 19;
END_IF


19:	(*Fördröj*)
fbDelay(IN:= TRUE, PT:=T#200MS , Q=> , ET=> );
IF fbDelay.Q THEN
	fbDelay(IN:= FALSE);
	nStat := 101;
END_IF;

101:(*ApparentPower*)
fbReadRegs(
					sIPAddr:= sSlaveIP,
					nTCPPort:= uiPort,
					nUnitID:= nUnit_ID,
					nQuantity:= 8,
					nMBAddr:= 30813 ,
					cbLength:= SIZEOF(stClusterCtrlData.stApparentPower) ,
					pDestAddr :=  ADR(stClusterCtrlData.stApparentPower),
					bExecute:= TRUE ,
					tTimeout:= T#2S ,bBusy=> ,	bError=> , nErrId=> ,cbRead=> );
					

IF fbReadRegs.bError THEN
	nStat := 999;
ELSIF  NOT fbReadRegs.bBusy AND NOT fbReadRegs.bError THEN
	fbReadRegs(bExecute := FALSE);
	nStat := 102;
END_IF


102:	(*Fördröj*)
fbDelay(IN:= TRUE, PT:=T#200MS , Q=> , ET=> );
IF fbDelay.Q THEN
	fbDelay(IN:= FALSE);
	nStat := 103;
END_IF;

103:(*nEnergySavingMode*)
fbReadRegs(
					sIPAddr:= sSlaveIP,
					nTCPPort:= uiPort,
					nUnitID:= nUnit_ID,
					nQuantity:= 2,
					nMBAddr:= 40695 ,
					cbLength:= SIZEOF(stClusterCtrlData.nEnergySavingMode) ,
					pDestAddr :=  ADR(stClusterCtrlData.nEnergySavingMode),
					bExecute:= TRUE ,
					tTimeout:= T#2S ,bBusy=> ,	bError=> , nErrId=> ,cbRead=> );					

IF fbReadRegs.bError THEN
	nStat := 999;
ELSIF  NOT fbReadRegs.bBusy AND NOT fbReadRegs.bError THEN
	fbReadRegs(bExecute := FALSE);
	nStat := 104;
END_IF

104:	(*Fördröj*)
fbDelay(IN:= TRUE, PT:=T#200MS , Q=> , ET=> );
IF fbDelay.Q THEN
	fbDelay(IN:= FALSE);
	nStat := 20;
END_IF;

20:(*Modbus Funktion 3, Läs data från Holding Registers*)
fbReadRegs(
					sIPAddr:= sSlaveIP,
					nTCPPort:= uiPort,
					nUnitID:= nUnit_ID2,
					nQuantity:= 8,
					nMBAddr:= 30775 ,
					cbLength:= SIZEOF(stClusterCtrlData2.stActivePower) ,
					pDestAddr :=  ADR(stClusterCtrlData2.stActivePower),
					bExecute:= TRUE ,
					tTimeout:= T#2S ,bBusy=> ,	bError=> , nErrId=> ,cbRead=> );
					

IF fbReadRegs.bError THEN
	nStat := 999;
ELSIF  NOT fbReadRegs.bBusy AND NOT fbReadRegs.bError THEN
	fbReadRegs(bExecute := FALSE);
	nStat := 21;
END_IF


21:	(*Fördröj*)
fbDelay(IN:= TRUE, PT:=T#200MS , Q=> , ET=> );
IF fbDelay.Q THEN
	fbDelay(IN:= FALSE);
	nStat := 22;
END_IF;


22:(*Modbus Funktion 3, Läs data från Holding Registers*)
fbReadRegs(
					sIPAddr:= sSlaveIP,
					nTCPPort:= uiPort,
					nUnitID:= nUnit_ID2,
					nQuantity:= 12,
					nMBAddr:= 30783 ,
					cbLength:= SIZEOF(stClusterCtrlData2.stLineVoltage) ,
					pDestAddr :=  ADR(stClusterCtrlData2.stLineVoltage),
					bExecute:= TRUE ,
					tTimeout:= T#2S ,bBusy=> ,	bError=> , nErrId=> ,cbRead=> );
					

IF fbReadRegs.bError THEN
	nStat := 999;
ELSIF  NOT fbReadRegs.bBusy AND NOT fbReadRegs.bError THEN
	fbReadRegs(bExecute := FALSE);
	nStat := 23;
END_IF


23:	(*Fördröj*)
fbDelay(IN:= TRUE, PT:=T#200MS , Q=> , ET=> );
IF fbDelay.Q THEN
	fbDelay(IN:= FALSE);
	nStat := 24;
END_IF;


24:(*Modbus Funktion 3, Läs data från Holding Registers*)
fbReadRegs(
					sIPAddr:= sSlaveIP,
					nTCPPort:= uiPort,
					nUnitID:= nUnit_ID2,
					nQuantity:= 10,
					nMBAddr:= 30795 ,
					cbLength:= SIZEOF(stClusterCtrlData2.stLineCurrent) ,
					pDestAddr :=  ADR(stClusterCtrlData2.stLineCurrent),
					bExecute:= TRUE ,
					tTimeout:= T#2S ,bBusy=> ,	bError=> , nErrId=> ,cbRead=> );
					

IF fbReadRegs.bError THEN
	nStat := 999;
ELSIF  NOT fbReadRegs.bBusy AND NOT fbReadRegs.bError THEN
	fbReadRegs(bExecute := FALSE);
	nStat := 25;
END_IF


25:	(*Fördröj*)
fbDelay(IN:= TRUE, PT:=T#200MS , Q=> , ET=> );
IF fbDelay.Q THEN
	fbDelay(IN:= FALSE);
	nStat := 26;
END_IF;


26:(*Modbus Funktion 3, Läs data från Holding Registers*)
fbReadRegs(
					sIPAddr:= sSlaveIP,
					nTCPPort:= uiPort,
					nUnitID:= nUnit_ID2,
					nQuantity:= 16,
					nMBAddr:= 30529 ,
					cbLength:= SIZEOF(stClusterCtrlData2.stYield) ,
					pDestAddr :=  ADR(stClusterCtrlData2.stYield),
					bExecute:= TRUE ,
					tTimeout:= T#2S ,bBusy=> ,	bError=> , nErrId=> ,cbRead=> );
					

IF fbReadRegs.bError THEN
	nStat := 999;
ELSIF  NOT fbReadRegs.bBusy AND NOT fbReadRegs.bError THEN
	fbReadRegs(bExecute := FALSE);
	nStat := 27;
END_IF


27:	(*Fördröj*)
fbDelay(IN:= TRUE, PT:=T#200MS , Q=> , ET=> );
IF fbDelay.Q THEN
	fbDelay(IN:= FALSE);
	nStat := 28;
END_IF;


28:(*Modbus Funktion 3, Läs data från Holding Registers*)
fbReadRegs(
					sIPAddr:= sSlaveIP,
					nTCPPort:= uiPort,
					nUnitID:= nUnit_ID2,
					nQuantity:= 8,
					nMBAddr:= 30977 ,
					cbLength:= SIZEOF(stClusterCtrlData2.stPVDATA) ,
					pDestAddr :=  ADR(stClusterCtrlData2.stPVDATA),
					bExecute:= TRUE ,
					tTimeout:= T#2S ,bBusy=> ,	bError=> , nErrId=> ,cbRead=> );
					

IF fbReadRegs.bError THEN
	nStat := 999;
ELSIF  NOT fbReadRegs.bBusy AND NOT fbReadRegs.bError THEN
	fbReadRegs(bExecute := FALSE);
	nStat := 29;
END_IF


29:	(*Fördröj*)
fbDelay(IN:= TRUE, PT:=T#200MS , Q=> , ET=> );
IF fbDelay.Q THEN
	fbDelay(IN:= FALSE);
	nStat := 30;
END_IF;


30:(*Modbus Funktion 3, Läs data från Holding Registers*)
fbReadRegs(
					sIPAddr:= sSlaveIP,
					nTCPPort:= uiPort,
					nUnitID:= nUnit_ID2,
					nQuantity:= 2,
					nMBAddr:= 30201 ,
					cbLength:= SIZEOF(stClusterCtrlData2.stStatus) ,
					pDestAddr :=  ADR(stClusterCtrlData2.stStatus),
					bExecute:= TRUE ,
					tTimeout:= T#2S ,bBusy=> ,	bError=> , nErrId=> ,cbRead=> );
					

IF fbReadRegs.bError THEN
	nStat := 999;
ELSIF  NOT fbReadRegs.bBusy AND NOT fbReadRegs.bError THEN
	fbReadRegs(bExecute := FALSE);
	nStat := 31;
END_IF


31:	(*Fördröj*)
fbDelay(IN:= TRUE, PT:=T#200MS , Q=> , ET=> );
IF fbDelay.Q THEN
	fbDelay(IN:= FALSE);
	nStat := 32;
END_IF;

32: (* nTotEnergyConsInternally *) 
fbReadRegs(
					sIPAddr:= sSlaveIP,
					nTCPPort:= uiPort,
					nUnitID:= nUnit_ID2,
					nQuantity:= 2,
					nMBAddr:= 30593 ,
					cbLength:= SIZEOF(stClusterCtrlData2.nTotEnergyConsInternally) ,
					pDestAddr :=  ADR(stClusterCtrlData2.nTotEnergyConsInternally),
					bExecute:= TRUE ,
					tTimeout:= T#2S ,bBusy=> ,	bError=> , nErrId=> ,cbRead=> );
					

IF fbReadRegs.bError THEN
	nStat := 999;
ELSIF  NOT fbReadRegs.bBusy AND NOT fbReadRegs.bError THEN
	fbReadRegs(bExecute := FALSE);
	nStat := 33;
END_IF

33:	(*Fördröj*)
fbDelay(IN:= TRUE, PT:=T#200MS , Q=> , ET=> );
IF fbDelay.Q THEN
	fbDelay(IN:= FALSE);
	nStat := 34;
END_IF;

34: (* nInverterInteriorTemp *) 
fbReadRegs(
					sIPAddr:= sSlaveIP,
					nTCPPort:= uiPort,
					nUnitID:= nUnit_ID2,
					nQuantity:= 2,
					nMBAddr:= 34113 ,
					cbLength:= SIZEOF(stClusterCtrlData2.nInverterInteriorTemp) ,
					pDestAddr :=  ADR(stClusterCtrlData2.nInverterInteriorTemp),
					bExecute:= TRUE ,
					tTimeout:= T#2S ,bBusy=> ,	bError=> , nErrId=> ,cbRead=> );
					

IF fbReadRegs.bError THEN
	nStat := 999;
ELSIF  NOT fbReadRegs.bBusy AND NOT fbReadRegs.bError THEN
	fbReadRegs(bExecute := FALSE);
	nStat := 35;
END_IF

35:	(*Fördröj*)
fbDelay(IN:= TRUE, PT:=T#200MS , Q=> , ET=> );
IF fbDelay.Q THEN
	fbDelay(IN:= FALSE);
	nStat := 36;
END_IF;	

36:(*ReactivePower*)
fbReadRegs(
					sIPAddr:= sSlaveIP,
					nTCPPort:= uiPort,
					nUnitID:= nUnit_ID2,
					nQuantity:= 8,
					nMBAddr:= 30805 ,
					cbLength:= SIZEOF(stClusterCtrlData2.stReactivePower) ,
					pDestAddr :=  ADR(stClusterCtrlData2.stReactivePower),
					bExecute:= TRUE ,
					tTimeout:= T#2S ,bBusy=> ,	bError=> , nErrId=> ,cbRead=> );
					
IF fbReadRegs.bError THEN
	nStat := 999;
ELSIF  NOT fbReadRegs.bBusy AND NOT fbReadRegs.bError THEN
	fbReadRegs(bExecute := FALSE);
	nStat := 37;
END_IF


37:	(*Fördröj*)
fbDelay(IN:= TRUE, PT:=T#200MS , Q=> , ET=> );
IF fbDelay.Q THEN
	fbDelay(IN:= FALSE);
	nStat := 38;
END_IF;

38:(*ApparentPower*)
fbReadRegs(
					sIPAddr:= sSlaveIP,
					nTCPPort:= uiPort,
					nUnitID:= nUnit_ID2,
					nQuantity:= 8,
					nMBAddr:= 30813 ,
					cbLength:= SIZEOF(stClusterCtrlData2.stApparentPower) ,
					pDestAddr :=  ADR(stClusterCtrlData2.stApparentPower),
					bExecute:= TRUE ,
					tTimeout:= T#2S ,bBusy=> ,	bError=> , nErrId=> ,cbRead=> );
					

IF fbReadRegs.bError THEN
	nStat := 999;
ELSIF  NOT fbReadRegs.bBusy AND NOT fbReadRegs.bError THEN
	fbReadRegs(bExecute := FALSE);
	nStat := 39;
END_IF


39:	(*Fördröj*)
fbDelay(IN:= TRUE, PT:=T#200MS , Q=> , ET=> );
IF fbDelay.Q THEN
	fbDelay(IN:= FALSE);
	nStat := 201;
END_IF;

201:(*nEnergySavingMode*)
fbReadRegs(
					sIPAddr:= sSlaveIP,
					nTCPPort:= uiPort,
					nUnitID:= nUnit_ID2,
					nQuantity:= 2,
					nMBAddr:= 40695 ,
					cbLength:= SIZEOF(stClusterCtrlData2.nEnergySavingMode) ,
					pDestAddr :=  ADR(stClusterCtrlData2.nEnergySavingMode),
					bExecute:= TRUE ,
					tTimeout:= T#2S ,bBusy=> ,	bError=> , nErrId=> ,cbRead=> );					

IF fbReadRegs.bError THEN
	nStat := 999;
ELSIF  NOT fbReadRegs.bBusy AND NOT fbReadRegs.bError THEN
	fbReadRegs(bExecute := FALSE);
	nStat := 202;
END_IF

202:	(*Fördröj*)
fbDelay(IN:= TRUE, PT:=T#200MS , Q=> , ET=> );
IF fbDelay.Q THEN
	fbDelay(IN:= FALSE);
	nStat := 40;
END_IF;



40:(*Modbus Funktion 3, Läs data från Holding Registers*)
fbReadRegs(
					sIPAddr:= sSlaveIP,
					nTCPPort:= uiPort,
					nUnitID:= nUnit_ID3,
					nQuantity:= 8,
					nMBAddr:= 30775 ,
					cbLength:= SIZEOF(stClusterCtrlData3.stActivePower) ,
					pDestAddr :=  ADR(stClusterCtrlData3.stActivePower),
					bExecute:= TRUE ,
					tTimeout:= T#2S ,bBusy=> ,	bError=> , nErrId=> ,cbRead=> );
					

IF fbReadRegs.bError THEN
	nStat := 999;
ELSIF  NOT fbReadRegs.bBusy AND NOT fbReadRegs.bError THEN
	fbReadRegs(bExecute := FALSE);
	nStat := 41;
END_IF


41:	(*Fördröj*)
fbDelay(IN:= TRUE, PT:=T#200MS , Q=> , ET=> );
IF fbDelay.Q THEN
	fbDelay(IN:= FALSE);
	nStat := 42;
END_IF;


42:(*Modbus Funktion 3, Läs data från Holding Registers*)
fbReadRegs(
					sIPAddr:= sSlaveIP,
					nTCPPort:= uiPort,
					nUnitID:= nUnit_ID3,
					nQuantity:= 12,
					nMBAddr:= 30783 ,
					cbLength:= SIZEOF(stClusterCtrlData3.stLineVoltage) ,
					pDestAddr :=  ADR(stClusterCtrlData3.stLineVoltage),
					bExecute:= TRUE ,
					tTimeout:= T#2S ,bBusy=> ,	bError=> , nErrId=> ,cbRead=> );
					

IF fbReadRegs.bError THEN
	nStat := 999;
ELSIF  NOT fbReadRegs.bBusy AND NOT fbReadRegs.bError THEN
	fbReadRegs(bExecute := FALSE);
	nStat := 43;
END_IF


43:	(*Fördröj*)
fbDelay(IN:= TRUE, PT:=T#200MS , Q=> , ET=> );
IF fbDelay.Q THEN
	fbDelay(IN:= FALSE);
	nStat := 44;
END_IF;


44:(*Modbus Funktion 3, Läs data från Holding Registers*)
fbReadRegs(
					sIPAddr:= sSlaveIP,
					nTCPPort:= uiPort,
					nUnitID:= nUnit_ID3,
					nQuantity:= 10,
					nMBAddr:= 30795 ,
					cbLength:= SIZEOF(stClusterCtrlData3.stLineCurrent) ,
					pDestAddr :=  ADR(stClusterCtrlData3.stLineCurrent),
					bExecute:= TRUE ,
					tTimeout:= T#2S ,bBusy=> ,	bError=> , nErrId=> ,cbRead=> );
					

IF fbReadRegs.bError THEN
	nStat := 999;
ELSIF  NOT fbReadRegs.bBusy AND NOT fbReadRegs.bError THEN
	fbReadRegs(bExecute := FALSE);
	nStat := 45;
END_IF


45:	(*Fördröj*)
fbDelay(IN:= TRUE, PT:=T#200MS , Q=> , ET=> );
IF fbDelay.Q THEN
	fbDelay(IN:= FALSE);
	nStat := 46;
END_IF;


46:(*Modbus Funktion 3, Läs data från Holding Registers*)
fbReadRegs(
					sIPAddr:= sSlaveIP,
					nTCPPort:= uiPort,
					nUnitID:= nUnit_ID3,
					nQuantity:= 16,
					nMBAddr:= 30529 ,
					cbLength:= SIZEOF(stClusterCtrlData3.stYield) ,
					pDestAddr :=  ADR(stClusterCtrlData3.stYield),
					bExecute:= TRUE ,
					tTimeout:= T#2S ,bBusy=> ,	bError=> , nErrId=> ,cbRead=> );
					

IF fbReadRegs.bError THEN
	nStat := 999;
ELSIF  NOT fbReadRegs.bBusy AND NOT fbReadRegs.bError THEN
	fbReadRegs(bExecute := FALSE);
	nStat := 47;
END_IF


47:	(*Fördröj*)
fbDelay(IN:= TRUE, PT:=T#200MS , Q=> , ET=> );
IF fbDelay.Q THEN
	fbDelay(IN:= FALSE);
	nStat := 48;
END_IF;


48:(*Modbus Funktion 3, Läs data från Holding Registers*)
fbReadRegs(
					sIPAddr:= sSlaveIP,
					nTCPPort:= uiPort,
					nUnitID:= nUnit_ID3,
					nQuantity:= 8,
					nMBAddr:= 30977 ,
					cbLength:= SIZEOF(stClusterCtrlData3.stPVDATA) ,
					pDestAddr :=  ADR(stClusterCtrlData3.stPVDATA),
					bExecute:= TRUE ,
					tTimeout:= T#2S ,bBusy=> ,	bError=> , nErrId=> ,cbRead=> );
					

IF fbReadRegs.bError THEN
	nStat := 999;
ELSIF  NOT fbReadRegs.bBusy AND NOT fbReadRegs.bError THEN
	fbReadRegs(bExecute := FALSE);
	nStat := 49;
END_IF


49:	(*Fördröj*)
fbDelay(IN:= TRUE, PT:=T#200MS , Q=> , ET=> );
IF fbDelay.Q THEN
	fbDelay(IN:= FALSE);
	nStat := 50;
END_IF;


50:(*Modbus Funktion 3, Läs data från Holding Registers*)
fbReadRegs(
					sIPAddr:= sSlaveIP,
					nTCPPort:= uiPort,
					nUnitID:= nUnit_ID3,
					nQuantity:= 2,
					nMBAddr:= 30201 ,
					cbLength:= SIZEOF(stClusterCtrlData3.stStatus) ,
					pDestAddr :=  ADR(stClusterCtrlData3.stStatus),
					bExecute:= TRUE ,
					tTimeout:= T#2S ,bBusy=> ,	bError=> , nErrId=> ,cbRead=> );
					

IF fbReadRegs.bError THEN
	nStat := 999;
ELSIF  NOT fbReadRegs.bBusy AND NOT fbReadRegs.bError THEN
	fbReadRegs(bExecute := FALSE);
	nStat := 51;
END_IF


51:	(*Fördröj*)
fbDelay(IN:= TRUE, PT:=T#200MS , Q=> , ET=> );
IF fbDelay.Q THEN
	fbDelay(IN:= FALSE);
	nStat := 52;
END_IF;

52: (* nTotEnergyConsInternally *) 
fbReadRegs(
					sIPAddr:= sSlaveIP,
					nTCPPort:= uiPort,
					nUnitID:= nUnit_ID3,
					nQuantity:= 2,
					nMBAddr:= 30593 ,
					cbLength:= SIZEOF(stClusterCtrlData3.nTotEnergyConsInternally) ,
					pDestAddr :=  ADR(stClusterCtrlData3.nTotEnergyConsInternally),
					bExecute:= TRUE ,
					tTimeout:= T#2S ,bBusy=> ,	bError=> , nErrId=> ,cbRead=> );
					

IF fbReadRegs.bError THEN
	nStat := 999;
ELSIF  NOT fbReadRegs.bBusy AND NOT fbReadRegs.bError THEN
	fbReadRegs(bExecute := FALSE);
	nStat := 53;
END_IF

53:	(*Fördröj*)
fbDelay(IN:= TRUE, PT:=T#200MS , Q=> , ET=> );
IF fbDelay.Q THEN
	fbDelay(IN:= FALSE);
	nStat := 54;
END_IF;

54: (* nInverterInteriorTemp *) 
fbReadRegs(
					sIPAddr:= sSlaveIP,
					nTCPPort:= uiPort,
					nUnitID:= nUnit_ID3,
					nQuantity:= 2,
					nMBAddr:= 34113 ,
					cbLength:= SIZEOF(stClusterCtrlData3.nInverterInteriorTemp) ,
					pDestAddr :=  ADR(stClusterCtrlData3.nInverterInteriorTemp),
					bExecute:= TRUE ,
					tTimeout:= T#2S ,bBusy=> ,	bError=> , nErrId=> ,cbRead=> );
					

IF fbReadRegs.bError THEN
	nStat := 999;
ELSIF  NOT fbReadRegs.bBusy AND NOT fbReadRegs.bError THEN
	fbReadRegs(bExecute := FALSE);
	nStat := 55;
END_IF

55:	(*Fördröj*)
fbDelay(IN:= TRUE, PT:=T#200MS , Q=> , ET=> );
IF fbDelay.Q THEN
	fbDelay(IN:= FALSE);
	nStat := 56;
END_IF;	

56:(*ReactivePower*)
fbReadRegs(
					sIPAddr:= sSlaveIP,
					nTCPPort:= uiPort,
					nUnitID:= nUnit_ID3,
					nQuantity:= 8,
					nMBAddr:= 30805 ,
					cbLength:= SIZEOF(stClusterCtrlData3.stReactivePower) ,
					pDestAddr :=  ADR(stClusterCtrlData3.stReactivePower),
					bExecute:= TRUE ,
					tTimeout:= T#2S ,bBusy=> ,	bError=> , nErrId=> ,cbRead=> );
					
IF fbReadRegs.bError THEN
	nStat := 999;
ELSIF  NOT fbReadRegs.bBusy AND NOT fbReadRegs.bError THEN
	fbReadRegs(bExecute := FALSE);
	nStat := 57;
END_IF


57:	(*Fördröj*)
fbDelay(IN:= TRUE, PT:=T#200MS , Q=> , ET=> );
IF fbDelay.Q THEN
	fbDelay(IN:= FALSE);
	nStat := 58;
END_IF;

58:(*ApparentPower*)
fbReadRegs(
					sIPAddr:= sSlaveIP,
					nTCPPort:= uiPort,
					nUnitID:= nUnit_ID3,
					nQuantity:= 8,
					nMBAddr:= 30813 ,
					cbLength:= SIZEOF(stClusterCtrlData3.stApparentPower) ,
					pDestAddr :=  ADR(stClusterCtrlData3.stApparentPower),
					bExecute:= TRUE ,
					tTimeout:= T#2S ,bBusy=> ,	bError=> , nErrId=> ,cbRead=> );
					

IF fbReadRegs.bError THEN
	nStat := 999;
ELSIF  NOT fbReadRegs.bBusy AND NOT fbReadRegs.bError THEN
	fbReadRegs(bExecute := FALSE);
	nStat := 59;
END_IF

59:	(*Fördröj*)
fbDelay(IN:= TRUE, PT:=T#200MS , Q=> , ET=> );
IF fbDelay.Q THEN
	fbDelay(IN:= FALSE);
	nStat := 60;
END_IF;

60:(*nEnergySavingMode*)
fbReadRegs(
					sIPAddr:= sSlaveIP,
					nTCPPort:= uiPort,
					nUnitID:= nUnit_ID3,
					nQuantity:= 2,
					nMBAddr:= 40695 ,
					cbLength:= SIZEOF(stClusterCtrlData3.nEnergySavingMode) ,
					pDestAddr :=  ADR(stClusterCtrlData3.nEnergySavingMode),
					bExecute:= TRUE ,
					tTimeout:= T#2S ,bBusy=> ,	bError=> , nErrId=> ,cbRead=> );
					

IF fbReadRegs.bError THEN
	nStat := 999;
ELSIF  NOT fbReadRegs.bBusy AND NOT fbReadRegs.bError THEN
	fbReadRegs(bExecute := FALSE);
	nStat := 61;
END_IF

61:	(*Fördröj*)
fbDelay(IN:= TRUE, PT:=T#200MS , Q=> , ET=> );
IF fbDelay.Q THEN
	fbDelay(IN:= FALSE);
	nStat := 62;
END_IF;

62:(*Si420TC*)
fbReadRegs(
					sIPAddr:= sSlaveIP,
					nTCPPort:= uiPort,
					nUnitID:= nUnit_ID3,
					nQuantity:= 4,
					nMBAddr:= 34623 ,
					cbLength:= SIZEOF(stClusterCtrlDataSensor.stSi420) , //Vet ej hur jag ska göra här
					pDestAddr :=  ADR(stClusterCtrlDataSensor.stSi420),
					bExecute:= TRUE ,
					tTimeout:= T#2S ,bBusy=> ,	bError=> , nErrId=> ,cbRead=> );
					

IF fbReadRegs.bError THEN
	nStat := 999;
ELSIF  NOT fbReadRegs.bBusy AND NOT fbReadRegs.bError THEN
	fbReadRegs(bExecute := FALSE);
	nStat := 63;
END_IF

63:	(*Fördröj*)
fbDelay(IN:= TRUE, PT:=T#200MS , Q=> , ET=> );
IF fbDelay.Q THEN
	fbDelay(IN:= FALSE);
	nStat := 0;
END_IF;



999:(*Något blev fel*)
	fbReadRegs(bExecute := FALSE);
	bCommErr:= TRUE;
	bBusy := FALSE;
	nStat := 0;
END_CASE

END_PROGRAM

// ---- POUs/_FBs/F_WordSwap.TcPOU
FUNCTION F_WordSwap : DWORD
VAR_INPUT
	nDataIn : DWORD;
END_VAR
VAR
	nHighWord : WORD;
	nLowWord : WORD;
END_VAR

nLowWord := DWORD_TO_WORD(nDataIn);
nHighWord := DWORD_TO_WORD( SHR(nDataIn, 16 ));

F_WordSwap := nHighWord + nLowWord;

END_FUNCTION

// ---- POUs/ClusterCtrl/F15_ClusterCtrl_Larm.TcPOU
PROGRAM F15_ClusterCtrl_Larm
VAR
	tof_0: TOF;

	FB_FL0: FB_FL;
	FB_FL1: FB_FL;
	FB_FL2: FB_FL;
	FB_FL3: FB_FL;
	FB_FL4: FB_FL;
	FB_FL5: FB_FL;
	FB_FL6: FB_FL;
	test: INT;
END_VAR
VAR // added by the converter: edge detectors and wires of the graphical bodies
    _w1, _w2 : ANY;
END_VAR

GVL_ClusterCtrl._CCtrl_V1_IT := _w1;
_w1 := F15_ClusterCtrl.DeviceStatus1 = 307;
GVL_Larm._CCtrl_V2_L := FB_FL3.Larm_ut;
GVL_ClusterCtrl._CCtrl_V2_IT := F15_ClusterCtrl.DeviceStatus2 = 307;
FB_FL1(Larm_in := _w2, TID_in := GVL_Larm._CCtrl_V1_L_FL); // FB_FL
FB_FL3(Larm_in := F15_ClusterCtrl.DeviceStatus2 = 35, TID_in := GVL_Larm._CCtrl_V2_L_FL); // FB_FL
tof_0(IN := ClusterControl_3Unit.bCommErr, PT := t#10S); // TOF
GVL_Larm._CCtrl_LC := FB_FL0.Larm_ut;
GVL_Larm._CCtrl_V2_LM := F15_ClusterCtrl.DeviceStatus2 = 303;
FB_FL0(Larm_in := tof_0.Q, TID_in := GVL_Larm._CCtrl_LC_FL); // FB_FL
_w2 := F15_ClusterCtrl.DeviceStatus1 = 35;
GVL_Larm._CCtrl_V1_L := FB_FL1.Larm_ut;
GVL_Larm._CCtrl_V1_LM := F15_ClusterCtrl.DeviceStatus1 = 303;
FB_FL5(Larm_in := F15_ClusterCtrl.DeviceStatus3 = 35, TID_in := GVL_Larm._CCtrl_V3_L_FL); // FB_FL
GVL_Larm._CCtrl_V3_L := FB_FL5.Larm_ut;
GVL_Larm._CCtrl_V3_LM := F15_ClusterCtrl.DeviceStatus3 = 303;
GVL_ClusterCtrl._CCtrl_V3_IT := F15_ClusterCtrl.DeviceStatus3 = 307;

END_PROGRAM

// ---- POUs/Systemprogram/PLC_Batteri_Larm.TcPOU
PROGRAM PLC_Batteri_Larm
VAR
	fbTime 						: FB_LocalSystemTime;	
	FB_Timesplit: FB_BA_ExtTiSt;
	FB_CountYears_0: FB_CountYears;

	TON_0: TON;
	TON_1: TON;
	
END_VAR

VAR PERSISTENT
	Years :DINT;
END_VAR
VAR // added by the converter: edge detectors and wires of the graphical bodies
    _w1, _w4 : BOOL;
    _w2, _w3, _w5 : ANY;
END_VAR

_w2 := _w1 OR TON_0.Q;
TON_0(IN := _w3, PT := T#60s); // TON
_w4 := PLC_TID.fbTime.systemTime.wMonth = 1 AND PLC_TID.fbTime.systemTime.wDay = 1 AND TON_1.Q;
_w1 := Years = 5;
GVL_Larm._BATT_L := _w2;
_w5 := GVL_Larm._BATT_L_ACK AND _w1;
TON_1(IN := TRUE, PT := t#5s); // TON
FB_CountYears_0(bCount := _w4, bReset := _w5, diYears := Years); // FB_CountYears
GVL_Larm._BATT_L_ACK := FALSE;
_w3 := PersistentData.FB_GetUPSStatus_0.stStatus.eBatteryStatus = 2;

END_PROGRAM

// ---- POUs/_FBs/FB_CountYears.TcPOU
FUNCTION_BLOCK FB_CountYears

(*Läser funktionsblock FB_Pulsfilter*)
VAR_INPUT
	bCount	: BOOL;
	bReset	:BOOL;

END_VAR

VAR_IN_OUT
	diYears	: DINT;

END_VAR

VAR
	pfReset	: R_TRIG;
	filterCount	: FB_Pulsfilter;

END_VAR

filterCount(bIN:=bCount,);
pfReset(CLK:= bReset,);


IF filterCount.bQ THEN
diYears := diYears + 1;
END_IF


IF pfReset.Q THEN
diYears := 0;
END_IF


IF bReset = TRUE THEN
bReset := FALSE;
END_IF

END_FUNCTION_BLOCK

// ---- POUs/_FBs/FB_Pulsfilter.TcPOU
FUNCTION_BLOCK FB_Pulsfilter

VAR_INPUT
	bIN: BOOL;
	FTimeOn: TIME:=t#2ms;
	FTimeOff: TIME:=t#2ms;
END_VAR
VAR_OUTPUT
	bQ: BOOL;
END_VAR
VAR

	FilterOn: TON;
	Pf_Trigg: R_TRIG;
	FilterOff: TOF;
	SetReset: SR;
END_VAR

FilterOn(IN:=bIN,);
FilterOn(PT:=FTimeOn,);
FilterOn.ET;

FilterOff(IN:=bIN,);
FilterOff(PT:=FTimeOff,);
FilterOff.ET;

SetReset(SET1:=FilterOn.Q,);
SetReset(RESET:=NOT FilterOff.Q,);

Pf_Trigg(CLK:=SetReset.Q1,);

IF Pf_Trigg.Q THEN
	bQ:=TRUE;
ELSE
	bQ:=FALSE;
END_IF

END_FUNCTION_BLOCK

// ---- POUs/Systemprogram/PLC_TID.TcPOU
PROGRAM PLC_TID
VAR
	fbTime 						: FB_LocalSystemTime; (*Function to get localsystemtime*)
	systemTime 					: T_MaxString;
END_VAR

(*Localsystemtime TimeStamp updater*)
fbTime(bEnable:=TRUE, dwCycle:= 1);
systemTime := SYSTEMTIME_TO_STRING(fbTime.systemTime);


GVL_IO._PLC_YY				:= fbTime.systemTime.wYear;
GVL_IO._PLC_MM				:= fbTime.systemTime.wMonth;
GVL_IO._PLC_DD				:= fbTime.systemTime.wDay;
GVL_IO._PLC_HHMM			:=(fbTime.systemTime.wHour)*100+(fbTime.systemTime.wMinute);

END_PROGRAM

// ---- POUs/Systemprogram/PersistentData.TcPOU
PROGRAM PersistentData
VAR
	
	FB_GetUPSStatus_0: FB_GetUPSStatus;
	FB_WritePersistent: FB_WritePersistentData;
	MODE :E_PersistentMode; 
	Status:ST_UPSStatus;
END_VAR
VAR // added by the converter: edge detectors and wires of the graphical bodies
    _w1 : BOOL;
    _w2 : ANY;
END_VAR

FB_GetUPSStatus_0(sNetId := '172.20.7.100.1.1', nPort := 0, bEnable := TRUE); // FB_GetUPSStatus
_w2 := FB_GetUPSStatus_0.bValid AND _w1;
_w1 := FB_GetUPSStatus_0.stStatus.ePowerStatus = 1;
FB_WritePersistent(NETID := '172.20.7.100.1.1', PORT := 852, START := NOT _w2, TMOUT := t#5s, MODE := MODE); // FB_WritePersistentData

END_PROGRAM

// ---- POUs/Loggning/MAIN_loggning.TcPOU
PROGRAM MAIN_loggning
VAR
	fbIoT : FB_IoT_Publisher;
END_VAR

(*Energimatare Schneider*)
IF GVL_Fastighet.CSVEnergyMeter THEN
	iEM3255_Logg();
END_IF

(*Cluster Control*)
IF GVL_Fastighet.CSVClusterCtrl THEN
	Cluster_Logg();
	Cluster_Logg_2();
	Cluster_Logg_3();
	Cluster_Sensor_Logg();
END_IF

(*Vaderstation*)
IF GVL_Fastighet.CSVWXT530 THEN
	WXT530_Logg();
END_IF

(*Temperaturgivare*)
IF GVL_Fastighet.CSVTempProbes THEN
	Temp_Logg();
END_IF
//SOLINSTRÅLNINGS MÄTARE
IF GVL_Fastighet.CSVSR05 THEN
	SR05_Logg();
END_IF

//IoT
fbIoT();

END_PROGRAM

// ---- POUs/Loggning/FB_IoT_Publisher.TcPOU
(*
 Library dependencies: Tc3_IotBase, Tc2_Utilities(3.3.21.0=>)
 License: TF6701
*)
FUNCTION_BLOCK FB_IoT_Publisher
VAR CONSTANT
	sEmptyString : STRING := '';
END_VAR
VAR_OUTPUT
	bActive : BOOL; (* FunctionBlock is executing *)
	bConnected : BOOL; (* Mqtt client is connected *)
	sErrorMsg : STRING;
	bError : BOOL; (* An Error is Active *)
	sLastPublishedTime : STRING; (* Timestamp of the last published message *)
	//nLastPublishedLength : INT; (* String length of the last published message *)
END_VAR
VAR
	(* Function Blocks *)	
		fbMqttClient : FB_IotMqttClient;
		fbTime 		 : FB_LocalSystemTime; (*Function to get localsystemtime*)	

	(* Mqtt specific *)	
		{attribute 'TcEncoding':='UTF-8'}
		sTopicPub : STRING(255);
		tPublishTime : TON;
		bConnect : BOOL;
		uPayload : U_Payload;
		sCurlyBracket : STRING := '{';
		sCurlyBracketEnd : STRING := '}';
		nPayloadLength : UINT;
		
	(* Local vars *)
		bInitDone : BOOL;
		sSystemTime : STRING(255);
		sJSONTime : STRING(255);
		nState : INT;
		i : INT;
		nPos : INT;
		nIteratorPackage : INT;
		
		//Remove
		bTest : BOOL;
		bTest1 : BOOL;
		hr : DINT;
		nCounter : INT;
END_VAR

//Call init the first plc-cycle only
IF NOT bInitDone THEN
	M_Initialize();
END_IF

//Update Queue Status
M_QueueBufferStatus();

//Update the system time
fbTime(bEnable:=TRUE, dwCycle:= 1);
sSystemTime := SYSTEMTIME_TO_STRING(fbTime.systemTime); 
sJSONTime := sSystemTime;
sJSONTime := REPLACE(sJSONTime, 'T', 1, 11);

//Execute the Mqtt Client
//The Execute()-method has to be called cyclically as background communication to the broker.
fbMqttClient.Execute(bConnect);

CASE nState OF

	0: (* Connect *)
		//Try to connect
		M_ConnectMQTT();
		
		//Check if connected
		IF fbMqttClient.bConnected THEN
			nState := 5;
		ELSIF bError THEN
			//Continue to fill the buffer and retry the connection
			nState := 10;
		END_IF
		
	5: (* Init *)
		bError := FALSE;
		sErrorMsg := '';
		tPublishTime(IN:=FALSE);
		nState := 10;		
		
	10: (* Build Payload *)
		tPublishTime(IN:=TRUE);
		IF tPublishTime.Q THEN
			
			IF nIteratorPackage >= 4 THEN
				M_CreatePayload(bFullPackage:=TRUE); //Build full package
				nIteratorPackage := 0;
			ELSIF nIteratorPackage < 4 THEN
				nIteratorPackage := nIteratorPackage + 1;
				M_CreatePayload(bFullPackage:=FALSE); //Build 'half' package
			END_IF			
			
			tPublishTime(IN:=FALSE);
			nState := 20;
		END_IF
			
	20: (* Publish *)
		IF fbMqttClient.bConnected THEN
			//Check if Buffer has messages
			IF NOT GVL_IoT.bBufferEmpty THEN
				M_Deque();
			END_IF
			
			//Then do a normal Publish
			M_Publish(uPayload);
			nState := 10; //Publish succeeded
		ELSE
			M_Queue(uPayload);
			nState := 600;
		END_IF

	600: (* Error State - Disconnect *)
		M_DisconnectMQTT();
		bError := TRUE;
		sErrorMsg := 'Lost connection to MQTT Client';
		
		nState := 0;

END_CASE

METHOD M_AddJSONObject
VAR_INPUT
	sObjectName : STRING;
	sObjectData : STRING;
END_VAR
VAR
	nStringPos : INT;
	sConcatMessage : STRING;
	sTempString : STRING := '';
	sEmpty : STRING;
	sDoubleQuote : STRING := '"';
	nStringLength : INT;
	sColon : STRING := ':';
	sComma : STRING := ',';
	nLastPos : UINT;
	i : UINT;
	x : INT;
	y : UINT;
END_VAR
//Check first empty position in the array
FOR i:=0 TO SIZEOF(uPayLoad.aPayload) / SIZEOF(uPayload.aPayload[0]) DO
	IF uPayload.aPayload[i] = 0 THEN
		nLastPos := nPayloadLength := i;
		EXIT;
	END_IF
END_FOR

//Check if empty
IF sObjectName <> '' AND sObjectData <> '' THEN

	IF sObjectName = 'Start' AND sObjectData = '{' THEN
		//Add the opening Curly Bracket '{'
		uPayload.aPayload[0] := ASC(sObjectData);
		
	ELSIF sObjectName = 'End' AND sObjectData = '}' THEN
		//Add the closing Curly Bracket '}' 
		// 44 = ',' in ASCII
		IF uPayload.aPayload[nLastPos - 1] = 44 THEN
			uPayload.aPayload[nLastPos - 1] := ASC(sObjectData);
		ELSE
			uPayload.aPayload[nLastPos] := ASC(sObjectData);
		END_IF
	ELSIF sObjectName = 'CollectionOpen' THEN
		//Add the following message: "objectData" : {
		sConcatMessage := CONCAT(sDoubleQuote,
						   CONCAT(sObjectData,
							CONCAT(sDoubleQuote,
						     CONCAT(sColon, '{'))));
								
		//Check the String length					 
		nStringLength := LEN(sConcatMessage);
		//Retrieve the last pos for the array to fill			
		y := nLastPos;
		//Loop trough every character in the string and convert it to ASCII code
		FOR x:=1 TO nStringLength DO
			sTempString := '';
			sTempString := MID(sConcatMessage,1,x);				
			uPayload.aPayload[y] := ASC(sTempString);
			y := y + 1;
		END_FOR
									
	ELSIF sObjectName = 'CollectionClose' THEN
		//Add the following message: },
		uPayload.aPayload[nLastPos - 1] := ASC('}');
		uPayload.aPayload[nLastPos] := ASC(sObjectData);		
	ELSE
		//Add the message (ObjectName + ObjectData)
		sTempString := sEmpty;

		// Add the following message: "objectName":"objectData",
		sConcatMessage := CONCAT(sDoubleQuote, 
							CONCAT(sObjectName,
							 CONCAT(sDoubleQuote,
							  CONCAT(sColon,
							   CONCAT(sDoubleQuote,
								CONCAT(sObjectData,
								 CONCAT(sDoubleQuote, sComma)))))));	
		//Check the String length					 
		nStringLength := LEN(sConcatMessage);
		//Retrieve the last pos for the array to fill			
		y := nLastPos;
		//Loop trough every character in the string and convert it to ASCII code
		FOR x:=1 TO nStringLength DO
			sTempString := '';
			sTempString := MID(sConcatMessage,1,x);				
			uPayload.aPayload[y] := ASC(sTempString);
			y := y + 1;
		END_FOR
		
	END_IF	
	
END_IF
END_METHOD

METHOD M_BuildPayload : BOOL
VAR_INPUT
	bFullPackage : BOOL;
END_VAR
// Method for building the Payload message that is going to be sent to the Azure IoT Hub. 
// Maximum 4kB message ANVÄNDS INTE GÖR CREATE BAYLOAD ISTÄLLET 
		
	//Clear Payload before creating a new one
	uPayload := GVL_IoT.uPayloadEmpty;
	
	//Build JSON-formatted string 
	//JSON Example: {"deviceId":"MyFirstDevice1","timeStamp":"2017-04-11T10:25:00.224"}	

	//Start Collection
	M_AddJSONObject('Start', sCurlyBracket);
	
	//Add your _Messages_ here:
	//////////////////////////////////////////
	//General
		M_AddJSONObject('ID', GVL_Fastighet.FastighetsBeteckning);
		M_AddJSONObject('timeStamp', sJSONTime);
	//Add new collection DataList
		M_AddJSONObject('CollectionOpen', 'DataList');
		
